KUKA KRL program: EPS_2_25694_WD05A_A_20260120031658.src

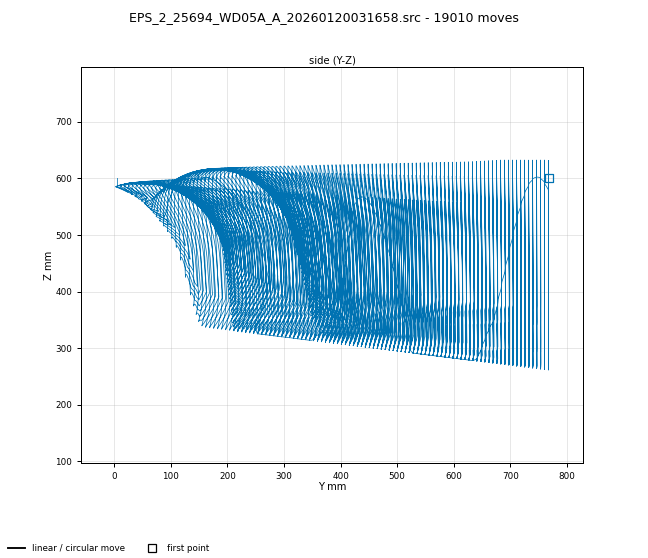
[picture p0: tool path of EPS_2_25694_WD05A_A_20260120031658.src, 19010 of 19012 moves have a stored position in this frame; points joined in program order, loops and branches not executed]
&ACCESS RVP
&REL 4
&COMMENT QRS 19112012
&PARAM EDITMASK = *
DEF PART()
EXT BAS (BAS_COMMAND :IN,REAL :IN )
INT I
BAS (#INITMOV,0 )

;KUKA QRS Post kuka4.cps  Date:22-06-2017 !

File_ID=3000

QRS_PRE_INIT()

;Init var - Until changes are made in qrs_pre_init
Outlet_Square_prg=0
Inlet_1_Square_prg=0
Inlet_2_Square_prg=0
Inlet_3_Square_prg=0
Inlet_4_Square_prg=0
Inlet_5_Square_prg=0

Outlet_1={X 0.000, Y 683.250, Z 507.000, B 0.000, E1 0.000 }
Inlet_1={X 0.000, Y 685.380, Z 477.000, B 0.000, E1 102.000 }
Inlet_2={X 0.000, Y 688.950, Z 427.000, B 0.000, E1 192.000 }
Outlet_1_type=251
Inlet_1_type=251
Inlet_2_type=251
;QRS#1=Sidecore dimensions
;QRS#2=250-10" PVC SDR 35
;QRS#3=250-10" PVC SDR 35
;QRS#4=250-10" PVC SDR 35
;QRS#5=
;QRS#6=
;QRS#7=
;QRS#8=
;QRS#9=14M PSX
;QRS#10=14M PSX
;QRS#11=14M PSX
;QRS#12=
;QRS#13=
;QRS#14=
;QRS#15=
;QRS#16=1524x152x991 3,25'
;QRS#17=EPS Height
;QRS#18=632,5
;QRS#19=*
;QRS#20= UPDATED VERSION 22-06-2017
;QRS#21=*
Outlet_Square=0100
Inlet_1_Square=0100
Inlet_2_Square=0100
Inlet_3_Square=0
Inlet_4_Square=0
Inlet_5_Square=0
Mill_Square=1
Outlet_Square_Prg=205
Inlet_1_Square_prg=205
Inlet_2_Square_prg=205

QRS_INIT()

$ADVANCE=5

; T1
PTP {E1 174.372,E2 174.372}
PTP {X 0,Y 767.508,A -85,B 0,C 180,E1 174.372,E2 174.372,E3 0,E4 0,E5 0,E6 0}
QRS_SPEED_INIT()
LIN {X 0,Y 767.508,Z 600,A -85,B 0,C 180,E1 174.372,E2 174.372,E3 0,E4 0,E5 0,E6 0} C_VEL
LIN {X 0,Y 767.508,Z 587.394,A -85,B 0,C 180,E1 174.372,E2 174.372} C_VEL
LIN {X 0,Y 767.508,Z 578.978,A -85,B 0,C 180,E1 174.372,E2 174.372} C_VEL
LIN {X 0,Y 767.496,Z 577.286,A -85,B 0,C 180,E1 174.143,E2 174.143} C_VEL
LIN {X 0,Y 767.495,Z 584.736,A -85,B 0,C 180,E1 173.186,E2 173.186} C_VEL
LIN {X 0,Y 767.498,Z 591.178,A -85,B 0,C 180,E1 172.132,E2 172.132} C_VEL
LIN {X 0,Y 767.492,Z 596.003,A -85,B 0,C 180,E1 171.075,E2 171.075} C_VEL
LIN {X 0,Y 767.497,Z 599.35,A -85,B 0,C 180,E1 170.014,E2 170.014} C_VEL
LIN {X 0,Y 767.492,Z 601.3,A -85,B 0,C 180,E1 168.951,E2 168.951} C_VEL
LIN {X 0,Y 767.498,Z 601.872,A -85,B 0,C 180,E1 167.883,E2 167.883} C_VEL
LIN {X 0,Y 767.495,Z 601.085,A -85,B 0,C 180,E1 166.811,E2 166.811} C_VEL
LIN {X 0,Y 767.497,Z 598.914,A -85,B 0,C 180,E1 165.735,E2 165.735} C_VEL
LIN {X 0,Y 767.496,Z 595.272,A -85,B 0,C 180,E1 164.653,E2 164.653} C_VEL
LIN {X 0,Y 767.496,Z 590.038,A -85,B 0,C 180,E1 163.566,E2 163.566} C_VEL
LIN {X 0,Y 767.497,Z 584.889,A -85,B 0,C 180,E1 162.746,E2 162.746} C_VEL
LIN {X 0,Y 767.497,Z 577.442,A -85,B 0,C 180,E1 161.786,E2 161.786} C_VEL
LIN {X 0,Y 767.497,Z 569.535,A -85,B 0,C 180,E1 160.958,E2 160.958} C_VEL
LIN {X 0,Y 767.498,Z 560.365,A -85,B 0,C 180,E1 160.16,E2 160.16} C_VEL
LIN {X 0,Y 767.498,Z 550.234,A -85,B 0,C 180,E1 159.429,E2 159.429} C_VEL
LIN {X 0,Y 767.498,Z 538.398,A -85,B 0,C 180,E1 158.729,E2 158.729} C_VEL
LIN {X 0,Y 767.475,Z 526.685,A -85,B 0,C 180,E1 158.163,E2 158.163} C_VEL
LIN {X 0,Y 767.49,Z 514.099,A -85,B 0,C 180,E1 157.673,E2 157.673} C_VEL
LIN {X 0,Y 767.495,Z 500.169,A -85,B 0,C 180,E1 157.255,E2 157.255} C_VEL
LIN {X 0,Y 767.49,Z 487.078,A -85,B 0,C 180,E1 156.967,E2 156.967} C_VEL
LIN {X 0,Y 767.49,Z 473.61,A -85,B 0,C 180,E1 156.769,E2 156.769} C_VEL
LIN {X 0,Y 767.47,Z 340.133,A -85,B 0,C 180,E1 155.5,E2 155.5} C_VEL
LIN {X 0,Y 767.459,Z 318.185,A -85,B 0,C 180,E1 153.141,E2 153.141} C_VEL
LIN {X 0,Y 767.478,Z 297.746,A -85,B 0,C 180,E1 150.923,E2 150.923} C_VEL
LIN {X 0,Y 767.488,Z 274.468,A -85,B 0,C 180,E1 148.366,E2 148.366} C_VEL
LIN {X 0,Y 767.445,Z 261.318,A -85,B 0,C 180,E1 146.893,E2 146.893} C_VEL
LIN {X 0,Y 767.439,Z 261.317,A -85,B 0,C 180,E1 144.9,E2 144.9} C_VEL
LIN {X 0,Y 767.432,Z 261.318,A -85,B 0,C 180,E1 142.959,E2 142.959} C_VEL
LIN {X 0,Y 767.427,Z 261.318,A -85,B 0,C 180,E1 140.879,E2 140.879} C_VEL
LIN {X 0,Y 767.421,Z 261.319,A -85,B 0,C 180,E1 138.916,E2 138.916} C_VEL
LIN {X 0,Y 767.423,Z 261.32,A -85,B 0,C 180,E1 136.8,E2 136.8} C_VEL
LIN {X 0,Y 767.441,Z 261.321,A -85,B 0,C 180,E1 134.61,E2 134.61} C_VEL
LIN {X 0,Y 767.488,Z 261.324,A -85,B 0,C 180,E1 132.333,E2 132.333} C_VEL
LIN {X 0,Y 767.43,Z 261.325,A -85,B 0,C 180,E1 129.943,E2 129.943} C_VEL
LIN {X 0,Y 767.411,Z 261.322,A -85,B 0,C 180,E1 127.701,E2 127.701} C_VEL
LIN {X 0,Y 767.415,Z 261.321,A -85,B 0,C 180,E1 125.676,E2 125.676} C_VEL
LIN {X 0,Y 767.426,Z 261.319,A -85,B 0,C 180,E1 123.833,E2 123.833} C_VEL
LIN {X 0,Y 767.433,Z 261.317,A -85,B 0,C 180,E1 121.916,E2 121.916} C_VEL
LIN {X 0,Y 767.433,Z 261.317,A -85,B 0,C 180,E1 119.879,E2 119.879} C_VEL
LIN {X 0,Y 767.438,Z 261.318,A -85,B 0,C 180,E1 117.709,E2 117.709} C_VEL
LIN {X 0,Y 767.47,Z 261.322,A -85,B 0,C 180,E1 115.373,E2 115.373} C_VEL
LIN {X 0,Y 767.49,Z 261.31,A -85,B 0,C 180,E1 112.814,E2 112.814} C_VEL
LIN {X 0,Y 767.465,Z 261.31,A -85,B 0,C 180,E1 110.294,E2 110.294} C_VEL
LIN {X 0,Y 767.463,Z 261.314,A -85,B 0,C 180,E1 108.079,E2 108.079} C_VEL
LIN {X 0,Y 767.477,Z 261.32,A -85,B 0,C 180,E1 105.891,E2 105.891} C_VEL
LIN {X 0,Y 767.491,Z 261.326,A -85,B 0,C 180,E1 103.728,E2 103.728} C_VEL
LIN {X 0,Y 767.477,Z 261.319,A -85,B 0,C 180,E1 101.584,E2 101.584} C_VEL
LIN {X 0,Y 767.466,Z 261.315,A -85,B 0,C 180,E1 99.457,E2 99.457} C_VEL
LIN {X 0,Y 767.463,Z 261.311,A -85,B 0,C 180,E1 97.342,E2 97.342} C_VEL
LIN {X 0,Y 767.466,Z 261.309,A -85,B 0,C 180,E1 95.238,E2 95.238} C_VEL
LIN {X 0,Y 767.488,Z 261.451,A -85,B 0,C 180,E1 94.68,E2 94.68} C_VEL
LIN {X 0,Y 767.448,Z 277.919,A -85,B 0,C 180,E1 92.355,E2 92.355} C_VEL
LIN {X 0,Y 767.478,Z 291.914,A -85,B 0,C 180,E1 90.393,E2 90.393} C_VEL
LIN {X 0,Y 767.487,Z 427.006,A -85,B 0,C 180,E1 89.103,E2 89.103} C_VEL
LIN {X 0,Y 767.496,Z 441.53,A -85,B 0,C 180,E1 88.857,E2 88.857} C_VEL
LIN {X 0,Y 767.491,Z 454.808,A -85,B 0,C 180,E1 88.53,E2 88.53} C_VEL
LIN {X 0,Y 767.491,Z 467.782,A -85,B 0,C 180,E1 88.105,E2 88.105} C_VEL
LIN {X 0,Y 767.489,Z 480.34,A -85,B 0,C 180,E1 87.582,E2 87.582} C_VEL
LIN {X 0,Y 767.499,Z 492.93,A -85,B 0,C 180,E1 86.928,E2 86.928} C_VEL
LIN {X 0,Y 767.497,Z 504.226,A -85,B 0,C 180,E1 86.208,E2 86.208} C_VEL
LIN {X 0,Y 767.496,Z 514.374,A -85,B 0,C 180,E1 85.421,E2 85.421} C_VEL
LIN {X 0,Y 767.498,Z 522.781,A -85,B 0,C 180,E1 84.634,E2 84.634} C_VEL
LIN {X 0,Y 767.497,Z 530.839,A -85,B 0,C 180,E1 83.714,E2 83.714} C_VEL
LIN {X 0,Y 767.498,Z 536.529,A -85,B 0,C 180,E1 82.924,E2 82.924} C_VEL
LIN {X 0,Y 767.499,Z 541.169,A -85,B 0,C 180,E1 82.133,E2 82.133} C_VEL
LIN {X 0,Y 767.498,Z 545.995,A -85,B 0,C 180,E1 81.076,E2 81.076} C_VEL
LIN {X 0,Y 767.493,Z 549.347,A -85,B 0,C 180,E1 80.016,E2 80.016} C_VEL
LIN {X 0,Y 767.491,Z 551.299,A -85,B 0,C 180,E1 78.952,E2 78.952} C_VEL
LIN {X 0,Y 767.497,Z 551.873,A -85,B 0,C 180,E1 77.885,E2 77.885} C_VEL
LIN {X 0,Y 767.495,Z 551.087,A -85,B 0,C 180,E1 76.813,E2 76.813} C_VEL
LIN {X 0,Y 767.49,Z 548.919,A -85,B 0,C 180,E1 75.736,E2 75.736} C_VEL
LIN {X 0,Y 767.492,Z 545.279,A -85,B 0,C 180,E1 74.654,E2 74.654} C_VEL
LIN {X 0,Y 767.496,Z 540.047,A -85,B 0,C 180,E1 73.567,E2 73.567} C_VEL
LIN {X 0,Y 767.498,Z 534.9,A -85,B 0,C 180,E1 72.748,E2 72.748} C_VEL
LIN {X 0,Y 767.497,Z 527.445,A -85,B 0,C 180,E1 71.786,E2 71.786} C_VEL
LIN {X 0,Y 767.496,Z 519.552,A -85,B 0,C 180,E1 70.959,E2 70.959} C_VEL
LIN {X 0,Y 767.498,Z 510.369,A -85,B 0,C 180,E1 70.16,E2 70.16} C_VEL
LIN {X 0,Y 767.498,Z 500.261,A -85,B 0,C 180,E1 69.431,E2 69.431} C_VEL
LIN {X 0,Y 767.498,Z 488.432,A -85,B 0,C 180,E1 68.731,E2 68.731} C_VEL
LIN {X 0,Y 767.482,Z 476.709,A -85,B 0,C 180,E1 68.164,E2 68.164} C_VEL
LIN {X 0,Y 767.474,Z 464.146,A -85,B 0,C 180,E1 67.675,E2 67.675} C_VEL
LIN {X 0,Y 767.496,Z 450.193,A -85,B 0,C 180,E1 67.255,E2 67.255} C_VEL
LIN {X 0,Y 767.466,Z 437.138,A -85,B 0,C 180,E1 66.968,E2 66.968} C_VEL
LIN {X 0,Y 767.451,Z 423.723,A -85,B 0,C 180,E1 66.77,E2 66.77} C_VEL
LIN {X 0,Y 767.496,Z 291.939,A -85,B 0,C 180,E1 65.521,E2 65.521} C_VEL
LIN {X 0,Y 767.491,Z 273.937,A -85,B 0,C 180,E1 62.997,E2 62.997} C_VEL
LIN {X 0,Y 767.45,Z 261.318,A -85,B 0,C 180,E1 61.185,E2 61.185} C_VEL
LIN {X 0,Y 767.434,Z 261.318,A -85,B 0,C 180,E1 59.087,E2 59.087} C_VEL
LIN {X 0,Y 767.412,Z 261.32,A -85,B 0,C 180,E1 56.797,E2 56.797} C_VEL
LIN {X 0,Y 767.416,Z 261.319,A -85,B 0,C 180,E1 54.901,E2 54.901} C_VEL
LIN {X 0,Y 767.417,Z 261.319,A -85,B 0,C 180,E1 52.96,E2 52.96} C_VEL
LIN {X 0,Y 767.413,Z 261.319,A -85,B 0,C 180,E1 50.88,E2 50.88} C_VEL
LIN {X 0,Y 767.414,Z 261.319,A -85,B 0,C 180,E1 48.918,E2 48.918} C_VEL
LIN {X 0,Y 767.411,Z 261.32,A -85,B 0,C 180,E1 46.902,E2 46.902} C_VEL
LIN {X 0,Y 767.44,Z 261.317,A -85,B 0,C 180,E1 45.352,E2 45.352} C_VEL
LIN {X 0,Y 767.424,Z 261.318,A -85,B 0,C 180,E1 43.2,E2 43.2} C_VEL
LIN {X 0,Y 767.417,Z 261.319,A -85,B 0,C 180,E1 41.084,E2 41.084} C_VEL
LIN {X 0,Y 767.416,Z 261.319,A -85,B 0,C 180,E1 39.034,E2 39.034} C_VEL
LIN {X 0,Y 767.416,Z 261.319,A -85,B 0,C 180,E1 37.042,E2 37.042} C_VEL
LIN {X 0,Y 767.426,Z 261.321,A -85,B 0,C 180,E1 34.774,E2 34.774} C_VEL
LIN {X 0,Y 767.448,Z 261.323,A -85,B 0,C 180,E1 32.581,E2 32.581} C_VEL
LIN {X 0,Y 767.48,Z 261.313,A -85,B 0,C 180,E1 29.89,E2 29.89} C_VEL
LIN {X 0,Y 767.446,Z 261.316,A -85,B 0,C 180,E1 27.714,E2 27.714} C_VEL
LIN {X 0,Y 767.422,Z 261.317,A -85,B 0,C 180,E1 25.37,E2 25.37} C_VEL
LIN {X 0,Y 767.439,Z 261.315,A -85,B 0,C 180,E1 23.678,E2 23.678} C_VEL
LIN {X 0,Y 767.471,Z 261.313,A -85,B 0,C 180,E1 21.974,E2 21.974} C_VEL
LIN {X 0,Y 767.44,Z 261.315,A -85,B 0,C 180,E1 19.737,E2 19.737} C_VEL
LIN {X 0,Y 767.423,Z 261.317,A -85,B 0,C 180,E1 17.53,E2 17.53} C_VEL
LIN {X 0,Y 767.449,Z 261.314,A -85,B 0,C 180,E1 15.891,E2 15.891} C_VEL
LIN {X 0,Y 767.429,Z 261.316,A -85,B 0,C 180,E1 13.728,E2 13.728} C_VEL
LIN {X 0,Y 767.47,Z 261.312,A -85,B 0,C 180,E1 12.117,E2 12.117} C_VEL
LIN {X 0,Y 767.449,Z 261.313,A -85,B 0,C 180,E1 9.986,E2 9.986} C_VEL
LIN {X 0,Y 767.435,Z 261.315,A -85,B 0,C 180,E1 7.869,E2 7.869} C_VEL
LIN {X 0,Y 767.425,Z 261.317,A -85,B 0,C 180,E1 5.762,E2 5.762} C_VEL
LIN {X 0,Y 767.463,Z 261.312,A -85,B 0,C 180,E1 4.187,E2 4.187} C_VEL
LIN {X 0,Y 767.447,Z 261.313,A -85,B 0,C 180,E1 2.092,E2 2.092} C_VEL
LIN {X 0,Y 767.438,Z 261.314,A -85,B 0,C 180,E1 0,E2 0} C_VEL
LIN {X 0,Y 767.431,Z 261.315,A -85,B 0,C 180,E1 -2.092,E2 -2.092} C_VEL
LIN {X 0,Y 767.428,Z 261.317,A -85,B 0,C 180,E1 -4.187,E2 -4.187} C_VEL
LIN {X 0,Y 767.43,Z 261.318,A -85,B 0,C 180,E1 -6.288,E2 -6.288} C_VEL
LIN {X 0,Y 767.436,Z 261.319,A -85,B 0,C 180,E1 -8.397,E2 -8.397} C_VEL
LIN {X 0,Y 767.448,Z 261.321,A -85,B 0,C 180,E1 -10.518,E2 -10.518} C_VEL
LIN {X 0,Y 767.495,Z 261.312,A -85,B 0,C 180,E1 -13.189,E2 -13.189} C_VEL
LIN {X 0,Y 767.483,Z 261.309,A -85,B 0,C 180,E1 -15.347,E2 -15.347} C_VEL
LIN {X 0,Y 767.455,Z 261.311,A -85,B 0,C 180,E1 -17.529,E2 -17.529} C_VEL
LIN {X 0,Y 767.432,Z 261.316,A -85,B 0,C 180,E1 -19.939,E2 -19.939} C_VEL
LIN {X 0,Y 767.433,Z 261.317,A -85,B 0,C 180,E1 -21.976,E2 -21.976} C_VEL
LIN {X 0,Y 767.447,Z 261.321,A -85,B 0,C 180,E1 -24.25,E2 -24.25} C_VEL
LIN {X 0,Y 767.484,Z 261.328,A -85,B 0,C 180,E1 -26.574,E2 -26.574} C_VEL
LIN {X 0,Y 767.496,Z 261.31,A -85,B 0,C 180,E1 -28.927,E2 -28.927} C_VEL
LIN {X 0,Y 767.453,Z 261.311,A -85,B 0,C 180,E1 -31.348,E2 -31.348} C_VEL
LIN {X 0,Y 767.464,Z 261.309,A -85,B 0,C 180,E1 -33.203,E2 -33.203} C_VEL
LIN {X 0,Y 767.472,Z 261.309,A -85,B 0,C 180,E1 -35.098,E2 -35.098} C_VEL
LIN {X 0,Y 767.441,Z 261.313,A -85,B 0,C 180,E1 -37.438,E2 -37.438} C_VEL
LIN {X 0,Y 767.437,Z 261.318,A -85,B 0,C 180,E1 -39.709,E2 -39.709} C_VEL
LIN {X 0,Y 767.442,Z 261.319,A -85,B 0,C 180,E1 -41.78,E2 -41.78} C_VEL
LIN {X 0,Y 767.454,Z 261.322,A -85,B 0,C 180,E1 -43.919,E2 -43.919} C_VEL
LIN {X 0,Y 767.482,Z 261.326,A -85,B 0,C 180,E1 -46.137,E2 -46.137} C_VEL
LIN {X 0,Y 767.468,Z 261.308,A -85,B 0,C 180,E1 -48.922,E2 -48.922} C_VEL
LIN {X 0,Y 767.459,Z 261.309,A -85,B 0,C 180,E1 -50.971,E2 -50.971} C_VEL
LIN {X 0,Y 767.457,Z 261.31,A -85,B 0,C 180,E1 -52.962,E2 -52.962} C_VEL
LIN {X 0,Y 767.44,Z 261.314,A -85,B 0,C 180,E1 -55.228,E2 -55.228} C_VEL
LIN {X 0,Y 767.445,Z 261.317,A -85,B 0,C 180,E1 -57.421,E2 -57.421} C_VEL
LIN {X 0,Y 767.481,Z 261.326,A -85,B 0,C 180,E1 -59.872,E2 -59.872} C_VEL
LIN {X 0,Y 767.487,Z 261.312,A -85,B 0,C 180,E1 -62.285,E2 -62.285} C_VEL
LIN {X 0,Y 767.472,Z 261.307,A -85,B 0,C 180,E1 -64.627,E2 -64.627} C_VEL
LIN {X 0,Y 767.448,Z 261.312,A -85,B 0,C 180,E1 -66.894,E2 -66.894} C_VEL
LIN {X 0,Y 767.444,Z 261.474,A -85,B 0,C 180,E1 -67.176,E2 -67.176} C_VEL
LIN {X 0,Y 767.477,Z 284.386,A -85,B 0,C 180,E1 -69.43,E2 -69.43} C_VEL
LIN {X 0,Y 767.461,Z 308.744,A -85,B 0,C 180,E1 -71.791,E2 -71.791} C_VEL
LIN {X 0,Y 767.489,Z 335.826,A -85,B 0,C 180,E1 -74.383,E2 -74.383} C_VEL
LIN {X 0,Y 767.49,Z 364.366,A -85,B 0,C 180,E1 -77.081,E2 -77.081} C_VEL
LIN {X 0,Y 767.489,Z 369.344,A -85,B 0,C 180,E1 -77.549,E2 -77.549} C_VEL
LIN {X 0,Y 767.475,Z 506.982,A -85,B 0,C 180,E1 -78.852,E2 -78.852} C_VEL
LIN {X 0,Y 767.49,Z 520.974,A -85,B 0,C 180,E1 -79.085,E2 -79.085} C_VEL
LIN {X 0,Y 767.479,Z 534.589,A -85,B 0,C 180,E1 -79.418,E2 -79.418} C_VEL
LIN {X 0,Y 767.474,Z 546.922,A -85,B 0,C 180,E1 -79.816,E2 -79.816} C_VEL
LIN {X 0,Y 767.483,Z 559.858,A -85,B 0,C 180,E1 -80.35,E2 -80.35} C_VEL
LIN {X 0,Y 767.499,Z 571.476,A -85,B 0,C 180,E1 -80.944,E2 -80.944} C_VEL
LIN {X 0,Y 767.496,Z 582.151,A -85,B 0,C 180,E1 -81.605,E2 -81.605} C_VEL
LIN {X 0,Y 767.498,Z 592.712,A -85,B 0,C 180,E1 -82.397,E2 -82.397} C_VEL
LIN {X 0,Y 767.497,Z 601.428,A -85,B 0,C 180,E1 -83.188,E2 -83.188} C_VEL
LIN {X 0,Y 767.496,Z 608.249,A -85,B 0,C 180,E1 -83.926,E2 -83.926} C_VEL
LIN {X 0,Y 767.497,Z 614.711,A -85,B 0,C 180,E1 -84.765,E2 -84.765} C_VEL
LIN {X 0,Y 767.494,Z 621.131,A -85,B 0,C 180,E1 -85.814,E2 -85.814} C_VEL
LIN {X 0,Y 767.496,Z 625.929,A -85,B 0,C 180,E1 -86.862,E2 -86.862} C_VEL
LIN {X 0,Y 767.496,Z 629.265,A -85,B 0,C 180,E1 -87.909,E2 -87.909} C_VEL
LIN {X 0,Y 767.497,Z 631.231,A -85,B 0,C 180,E1 -88.955,E2 -88.955} C_VEL
LIN {X 0,Y 767.494,Z 631.889,A -85,B 0,C 180,E1 -90.001,E2 -90.001} C_VEL
LIN {X 0,Y 767.497,Z 631.228,A -85,B 0,C 180,E1 -91.047,E2 -91.047} C_VEL
LIN {X 0,Y 767.496,Z 629.258,A -85,B 0,C 180,E1 -92.093,E2 -92.093} C_VEL
LIN {X 0,Y 767.496,Z 625.919,A -85,B 0,C 180,E1 -93.14,E2 -93.14} C_VEL
LIN {X 0,Y 767.494,Z 621.118,A -85,B 0,C 180,E1 -94.188,E2 -94.188} C_VEL
LIN {X 0,Y 767.497,Z 614.693,A -85,B 0,C 180,E1 -95.237,E2 -95.237} C_VEL
LIN {X 0,Y 767.496,Z 608.238,A -85,B 0,C 180,E1 -96.075,E2 -96.075} C_VEL
LIN {X 0,Y 767.498,Z 600.054,A -85,B 0,C 180,E1 -96.947,E2 -96.947} C_VEL
LIN {X 0,Y 767.497,Z 591.068,A -85,B 0,C 180,E1 -97.737,E2 -97.737} C_VEL
LIN {X 0,Y 767.498,Z 580.173,A -85,B 0,C 180,E1 -98.53,E2 -98.53} C_VEL
LIN {X 0,Y 767.498,Z 569.055,A -85,B 0,C 180,E1 -99.191,E2 -99.191} C_VEL
LIN {X 0,Y 767.494,Z 556.885,A -85,B 0,C 180,E1 -99.783,E2 -99.783} C_VEL
LIN {X 0,Y 767.472,Z 544.967,A -85,B 0,C 180,E1 -100.253,E2 -100.253} C_VEL
LIN {X 0,Y 767.484,Z 532.071,A -85,B 0,C 180,E1 -100.651,E2 -100.651} C_VEL
LIN {X 0,Y 767.487,Z 519.13,A -85,B 0,C 180,E1 -100.951,E2 -100.951} C_VEL
LIN {X 0,Y 767.474,Z 505.285,A -85,B 0,C 180,E1 -101.167,E2 -101.167} C_VEL
LIN {X 0,Y 767.488,Z 369.199,A -85,B 0,C 180,E1 -102.465,E2 -102.465} C_VEL
LIN {X 0,Y 767.498,Z 342.937,A -85,B 0,C 180,E1 -104.942,E2 -104.942} C_VEL
LIN {X 0,Y 767.479,Z 315.807,A -85,B 0,C 180,E1 -107.529,E2 -107.529} C_VEL
LIN {X 0,Y 767.465,Z 289.028,A -85,B 0,C 180,E1 -110.117,E2 -110.117} C_VEL
LIN {X 0,Y 767.459,Z 264.333,A -85,B 0,C 180,E1 -112.541,E2 -112.541} C_VEL
LIN {X 0,Y 767.444,Z 261.317,A -85,B 0,C 180,E1 -112.844,E2 -112.844} C_VEL
LIN {X 0,Y 767.44,Z 261.316,A -85,B 0,C 180,E1 -114.826,E2 -114.826} C_VEL
LIN {X 0,Y 767.442,Z 261.319,A -85,B 0,C 180,E1 -116.567,E2 -116.567} C_VEL
LIN {X 0,Y 767.45,Z 261.321,A -85,B 0,C 180,E1 -118.334,E2 -118.334} C_VEL
LIN {X 0,Y 767.461,Z 261.323,A -85,B 0,C 180,E1 -120.132,E2 -120.132} C_VEL
LIN {X 0,Y 767.471,Z 261.324,A -85,B 0,C 180,E1 -121.962,E2 -121.962} C_VEL
LIN {X 0,Y 767.47,Z 261.325,A -85,B 0,C 180,E1 -123.847,E2 -123.847} C_VEL
LIN {X 0,Y 767.478,Z 261.325,A -85,B 0,C 180,E1 -125.74,E2 -125.74} C_VEL
LIN {X 0,Y 767.469,Z 261.325,A -85,B 0,C 180,E1 -127.698,E2 -127.698} C_VEL
LIN {X 0,Y 767.422,Z 261.324,A -85,B 0,C 180,E1 -129.942,E2 -129.942} C_VEL
LIN {X 0,Y 767.427,Z 261.325,A -85,B 0,C 180,E1 -131.782,E2 -131.782} C_VEL
LIN {X 0,Y 767.405,Z 261.325,A -85,B 0,C 180,E1 -133.923,E2 -133.923} C_VEL
LIN {X 0,Y 767.401,Z 261.323,A -85,B 0,C 180,E1 -136.077,E2 -136.077} C_VEL
LIN {X 0,Y 767.406,Z 261.323,A -85,B 0,C 180,E1 -138.218,E2 -138.218} C_VEL
LIN {X 0,Y 767.411,Z 261.321,A -85,B 0,C 180,E1 -140.059,E2 -140.059} C_VEL
LIN {X 0,Y 767.426,Z 261.319,A -85,B 0,C 180,E1 -141.716,E2 -141.716} C_VEL
LIN {X 0,Y 767.434,Z 261.317,A -85,B 0,C 180,E1 -143.611,E2 -143.611} C_VEL
LIN {X 0,Y 767.44,Z 261.315,A -85,B 0,C 180,E1 -145.537,E2 -145.537} C_VEL
LIN {X 0,Y 767.449,Z 261.314,A -85,B 0,C 180,E1 -147.419,E2 -147.419} C_VEL
LIN {X 0,Y 767.465,Z 261.311,A -85,B 0,C 180,E1 -149.263,E2 -149.263} C_VEL
LIN {X 0,Y 767.472,Z 261.309,A -85,B 0,C 180,E1 -151.183,E2 -151.183} C_VEL
LIN {X 0,Y 767.45,Z 261.312,A -85,B 0,C 180,E1 -153.437,E2 -153.437} C_VEL
LIN {X 0,Y 767.451,Z 261.318,A -85,B 0,C 180,E1 -155.751,E2 -155.751} C_VEL
LIN {X 0,Y 767.483,Z 261.323,A -85,B 0,C 180,E1 -158.026,E2 -158.026} C_VEL
LIN {X 0,Y 767.487,Z 261.319,A -85,B 0,C 180,E1 -160.264,E2 -160.264} C_VEL
LIN {X 0,Y 767.48,Z 261.311,A -85,B 0,C 180,E1 -162.472,E2 -162.472} C_VEL
LIN {X 0,Y 767.491,Z 261.304,A -85,B 0,C 180,E1 -164.653,E2 -164.653} C_VEL
LIN {X 0,Y 767.489,Z 261.303,A -85,B 0,C 180,E1 -166.811,E2 -166.811} C_VEL
LIN {X 0,Y 767.481,Z 261.322,A -85,B 0,C 180,E1 -169.483,E2 -169.483} C_VEL
LIN {X 0,Y 767.478,Z 261.447,A -85,B 0,C 180,E1 -171.008,E2 -171.008} C_VEL
LIN {X 0,Y 767.457,Z 283.481,A -85,B 0,C 180,E1 -173.449,E2 -173.449} C_VEL
LIN {X 0,Y 767.459,Z 303.894,A -85,B 0,C 180,E1 -175.682,E2 -175.682} C_VEL
LIN {X 0,Y 767.479,Z 326.891,A -85,B 0,C 180,E1 -178.169,E2 -178.169} C_VEL
LIN {X 0,Y 767.492,Z 340.14,A -85,B 0,C 180,E1 -179.591,E2 -179.591} C_VEL
LIN {X 0,Y 767.473,Z 477.124,A -85,B 0,C 180,E1 -180.899,E2 -180.899} C_VEL
LIN {X 0,Y 767.479,Z 491.605,A -85,B 0,C 180,E1 -181.144,E2 -181.144} C_VEL
LIN {X 0,Y 767.493,Z 504.85,A -85,B 0,C 180,E1 -181.471,E2 -181.471} C_VEL
LIN {X 0,Y 767.473,Z 517.827,A -85,B 0,C 180,E1 -181.896,E2 -181.896} C_VEL
LIN {X 0,Y 767.487,Z 530.368,A -85,B 0,C 180,E1 -182.419,E2 -182.419} C_VEL
LIN {X 0,Y 767.499,Z 542.953,A -85,B 0,C 180,E1 -183.073,E2 -183.073} C_VEL
LIN {X 0,Y 767.497,Z 554.246,A -85,B 0,C 180,E1 -183.794,E2 -183.794} C_VEL
LIN {X 0,Y 767.496,Z 564.389,A -85,B 0,C 180,E1 -184.58,E2 -184.58} C_VEL
LIN {X 0,Y 767.498,Z 572.794,A -85,B 0,C 180,E1 -185.368,E2 -185.368} C_VEL
LIN {X 0,Y 767.496,Z 577.286,A -85,B 0,C 180,E1 -185.857,E2 -185.857} C_VEL
LIN {X 0,Y 766.835,Z 580.572,A -85,B 0,C 180,E1 -186.229,E2 -186.229} C_VEL
LIN {X 0,Y 763.971,Z 585.532,A -85,B 0,C 180,E1 -186.84,E2 -186.84} C_VEL
LIN {X 0,Y 761.109,Z 589.729,A -85,B 0,C 180,E1 -187.476,E2 -187.476} C_VEL
LIN {X 0,Y 760.438,Z 591.975,A -85,B 0,C 180,E1 -187.881,E2 -187.881} C_VEL
LIN {X 0,Y 760.444,Z 595.945,A -85,B 0,C 180,E1 -188.742,E2 -188.742} C_VEL
LIN {X 0,Y 760.422,Z 599.305,A -85,B 0,C 180,E1 -189.731,E2 -189.731} C_VEL
LIN {X 0,Y 760.417,Z 601.287,A -85,B 0,C 180,E1 -190.616,E2 -190.616} C_VEL
LIN {X 0,Y 760.446,Z 602.402,A -85,B 0,C 180,E1 -191.691,E2 -191.691} C_VEL
LIN {X 0,Y 760.439,Z 602.159,A -85,B 0,C 180,E1 -192.772,E2 -192.772} C_VEL
LIN {X 0,Y 760.42,Z 600.537,A -85,B 0,C 180,E1 -193.857,E2 -193.857} C_VEL
LIN {X 0,Y 760.447,Z 597.472,A -85,B 0,C 180,E1 -194.946,E2 -194.946} C_VEL
LIN {X 0,Y 760.431,Z 592.858,A -85,B 0,C 180,E1 -196.042,E2 -196.042} C_VEL
LIN {X 0,Y 760.448,Z 588.36,A -85,B 0,C 180,E1 -196.844,E2 -196.844} C_VEL
LIN {X 0,Y 760.456,Z 581.463,A -85,B 0,C 180,E1 -197.834,E2 -197.834} C_VEL
LIN {X 0,Y 760.447,Z 572.963,A -85,B 0,C 180,E1 -198.807,E2 -198.807} C_VEL
LIN {X 0,Y 760.456,Z 563.937,A -85,B 0,C 180,E1 -199.645,E2 -199.645} C_VEL
LIN {X 0,Y 760.486,Z 554.782,A -85,B 0,C 180,E1 -200.356,E2 -200.356} C_VEL
LIN {X 0,Y 760.473,Z 544.026,A -85,B 0,C 180,E1 -201.052,E2 -201.052} C_VEL
LIN {X 0,Y 760.488,Z 532.055,A -85,B 0,C 180,E1 -201.689,E2 -201.689} C_VEL
LIN {X 0,Y 760.5,Z 518.772,A -85,B 0,C 180,E1 -202.258,E2 -202.258} C_VEL
LIN {X 0,Y 760.523,Z 506.057,A -85,B 0,C 180,E1 -202.685,E2 -202.685} C_VEL
LIN {X 0,Y 760.539,Z 491.807,A -85,B 0,C 180,E1 -203.045,E2 -203.045} C_VEL
LIN {X 0,Y 760.549,Z 477.909,A -85,B 0,C 180,E1 -203.284,E2 -203.284} C_VEL
LIN {X 0,Y 760.452,Z 340.316,A -85,B 0,C 180,E1 -204.614,E2 -204.614} C_VEL
LIN {X 0,Y 760.453,Z 318.478,A -85,B 0,C 180,E1 -206.977,E2 -206.977} C_VEL
LIN {X 0,Y 760.497,Z 299.436,A -85,B 0,C 180,E1 -209.058,E2 -209.058} C_VEL
LIN {X 0,Y 760.532,Z 277.263,A -85,B 0,C 180,E1 -211.511,E2 -211.511} C_VEL
LIN {X 0,Y 760.433,Z 262.316,A -85,B 0,C 180,E1 -213.203,E2 -213.203} C_VEL
LIN {X 0,Y 760.421,Z 262.315,A -85,B 0,C 180,E1 -215.472,E2 -215.472} C_VEL
LIN {X 0,Y 760.447,Z 262.313,A -85,B 0,C 180,E1 -217.613,E2 -217.613} C_VEL
LIN {X 0,Y 760.454,Z 262.323,A -85,B 0,C 180,E1 -220.148,E2 -220.148} C_VEL
LIN {X 0,Y 760.417,Z 262.318,A -85,B 0,C 180,E1 -222.531,E2 -222.531} C_VEL
LIN {X 0,Y 760.393,Z 262.321,A -85,B 0,C 180,E1 -224.434,E2 -224.434} C_VEL
LIN {X 0,Y 760.393,Z 262.318,A -85,B 0,C 180,E1 -226.695,E2 -226.695} C_VEL
LIN {X 0,Y 760.397,Z 262.318,A -85,B 0,C 180,E1 -228.452,E2 -228.452} C_VEL
LIN {X 0,Y 760.369,Z 262.321,A -85,B 0,C 180,E1 -230.696,E2 -230.696} C_VEL
LIN {X 0,Y 760.375,Z 262.32,A -85,B 0,C 180,E1 -232.555,E2 -232.555} C_VEL
LIN {X 0,Y 760.387,Z 262.319,A -85,B 0,C 180,E1 -234.525,E2 -234.525} C_VEL
LIN {X 0,Y 760.442,Z 262.318,A -85,B 0,C 180,E1 -236.951,E2 -236.951} C_VEL
LIN {X 0,Y 760.433,Z 262.317,A -85,B 0,C 180,E1 -239.561,E2 -239.561} C_VEL
LIN {X 0,Y 760.426,Z 262.314,A -85,B 0,C 180,E1 -241.98,E2 -241.98} C_VEL
LIN {X 0,Y 760.445,Z 262.312,A -85,B 0,C 180,E1 -243.759,E2 -243.759} C_VEL
LIN {X 0,Y 760.418,Z 262.316,A -85,B 0,C 180,E1 -246.089,E2 -246.089} C_VEL
LIN {X 0,Y 760.451,Z 262.32,A -85,B 0,C 180,E1 -248.482,E2 -248.482} C_VEL
LIN {X 0,Y 760.454,Z 262.321,A -85,B 0,C 180,E1 -250.634,E2 -250.634} C_VEL
LIN {X 0,Y 760.463,Z 262.314,A -85,B 0,C 180,E1 -252.857,E2 -252.857} C_VEL
LIN {X 0,Y 760.488,Z 262.306,A -85,B 0,C 180,E1 -255.262,E2 -255.262} C_VEL
LIN {X 0,Y 760.471,Z 262.313,A -85,B 0,C 180,E1 -257.768,E2 -257.768} C_VEL
LIN {X 0,Y 760.457,Z 262.318,A -85,B 0,C 180,E1 -260.251,E2 -260.251} C_VEL
LIN {X 0,Y 760.433,Z 262.314,A -85,B 0,C 180,E1 -262.59,E2 -262.59} C_VEL
LIN {X 0,Y 760.442,Z 262.312,A -85,B 0,C 180,E1 -264.714,E2 -264.714} C_VEL
LIN {X 0,Y 760.483,Z 262.368,A -85,B 0,C 180,E1 -265.277,E2 -265.277} C_VEL
LIN {X 0,Y 760.434,Z 280.746,A -85,B 0,C 180,E1 -267.887,E2 -267.887} C_VEL
LIN {X 0,Y 760.455,Z 292.23,A -85,B 0,C 180,E1 -269.504,E2 -269.504} C_VEL
LIN {X 0,Y 760.533,Z 428.035,A -85,B 0,C 180,E1 -270.807,E2 -270.807} C_VEL
LIN {X 0,Y 760.546,Z 442.227,A -85,B 0,C 180,E1 -271.054,E2 -271.054} C_VEL
LIN {X 0,Y 760.505,Z 456.48,A -85,B 0,C 180,E1 -271.417,E2 -271.417} C_VEL
LIN {X 0,Y 760.501,Z 469.136,A -85,B 0,C 180,E1 -271.846,E2 -271.846} C_VEL
LIN {X 0,Y 760.491,Z 481.494,A -85,B 0,C 180,E1 -272.374,E2 -272.374} C_VEL
LIN {X 0,Y 760.474,Z 493.961,A -85,B 0,C 180,E1 -273.035,E2 -273.035} C_VEL
LIN {X 0,Y 760.461,Z 504.215,A -85,B 0,C 180,E1 -273.695,E2 -273.695} C_VEL
LIN {X 0,Y 760.478,Z 514.465,A -85,B 0,C 180,E1 -274.489,E2 -274.489} C_VEL
LIN {X 0,Y 760.445,Z 522.969,A -85,B 0,C 180,E1 -275.284,E2 -275.284} C_VEL
LIN {X 0,Y 760.452,Z 531.026,A -85,B 0,C 180,E1 -276.199,E2 -276.199} C_VEL
LIN {X 0,Y 760.443,Z 537.724,A -85,B 0,C 180,E1 -277.142,E2 -277.142} C_VEL
LIN {X 0,Y 760.445,Z 543.596,A -85,B 0,C 180,E1 -278.207,E2 -278.207} C_VEL
LIN {X 0,Y 760.448,Z 547.001,A -85,B 0,C 180,E1 -279.007,E2 -279.007} C_VEL
LIN {X 0,Y 760.421,Z 550.213,A -85,B 0,C 180,E1 -280.078,E2 -280.078} C_VEL
LIN {X 0,Y 760.432,Z 552.012,A -85,B 0,C 180,E1 -281.152,E2 -281.152} C_VEL
LIN {X 0,Y 760.43,Z 552.452,A -85,B 0,C 180,E1 -282.23,E2 -282.23} C_VEL
LIN {X 0,Y 760.43,Z 551.525,A -85,B 0,C 180,E1 -283.312,E2 -283.312} C_VEL
LIN {X 0,Y 760.419,Z 549.195,A -85,B 0,C 180,E1 -284.399,E2 -284.399} C_VEL
LIN {X 0,Y 760.449,Z 545.375,A -85,B 0,C 180,E1 -285.491,E2 -285.491} C_VEL
LIN {X 0,Y 760.441,Z 541.411,A -85,B 0,C 180,E1 -286.314,E2 -286.314} C_VEL
LIN {X 0,Y 760.431,Z 536.46,A -85,B 0,C 180,E1 -287.141,E2 -287.141} C_VEL
LIN {X 0,Y 760.446,Z 529.22,A -85,B 0,C 180,E1 -288.11,E2 -288.11} C_VEL
LIN {X 0,Y 760.464,Z 521.562,A -85,B 0,C 180,E1 -288.944,E2 -288.944} C_VEL
LIN {X 0,Y 760.452,Z 512.245,A -85,B 0,C 180,E1 -289.784,E2 -289.784} C_VEL
LIN {X 0,Y 760.47,Z 501.87,A -85,B 0,C 180,E1 -290.556,E2 -290.556} C_VEL
LIN {X 0,Y 760.481,Z 490.379,A -85,B 0,C 180,E1 -291.262,E2 -291.262} C_VEL
LIN {X 0,Y 760.476,Z 477.5,A -85,B 0,C 180,E1 -291.901,E2 -291.901} C_VEL
LIN {X 0,Y 760.484,Z 464.93,A -85,B 0,C 180,E1 -292.399,E2 -292.399} C_VEL
LIN {X 0,Y 760.534,Z 451.893,A -85,B 0,C 180,E1 -292.803,E2 -292.803} C_VEL
LIN {X 0,Y 760.497,Z 438.047,A -85,B 0,C 180,E1 -293.12,E2 -293.12} C_VEL
LIN {X 0,Y 760.499,Z 424.267,A -85,B 0,C 180,E1 -293.329,E2 -293.329} C_VEL
LIN {X 0,Y 760.481,Z 292.176,A -85,B 0,C 180,E1 -294.593,E2 -294.593} C_VEL
LIN {X 0,Y 760.476,Z 274.24,A -85,B 0,C 180,E1 -297.123,E2 -297.123} C_VEL
LIN {X 0,Y 760.426,Z 262.317,A -85,B 0,C 180,E1 -298.831,E2 -298.831} C_VEL
LIN {X 0,Y 760.402,Z 262.317,A -85,B 0,C 180,E1 -301.055,E2 -301.055} C_VEL
LIN {X 0,Y 760.409,Z 262.316,A -85,B 0,C 180,E1 -303.045,E2 -303.045} C_VEL
LIN {X 0,Y 760.4,Z 262.317,A -85,B 0,C 180,E1 -304.933,E2 -304.933} C_VEL
LIN {X 0,Y 760.422,Z 262.316,A -85,B 0,C 180,E1 -306.777,E2 -306.777} C_VEL
LIN {X 0,Y 760.423,Z 262.315,A -85,B 0,C 180,E1 -308.78,E2 -308.78} C_VEL
LIN {X 0,Y 760.412,Z 262.315,A -85,B 0,C 180,E1 -310.946,E2 -310.946} C_VEL
LIN {X 0,Y 760.398,Z 262.317,A -85,B 0,C 180,E1 -312.97,E2 -312.97} C_VEL
LIN {X 0,Y 760.401,Z 262.316,A -85,B 0,C 180,E1 -315.174,E2 -315.174} C_VEL
LIN {X 0,Y 760.416,Z 262.318,A -85,B 0,C 180,E1 -317.466,E2 -317.466} C_VEL
LIN {X 0,Y 760.453,Z 262.322,A -85,B 0,C 180,E1 -319.86,E2 -319.86} C_VEL
LIN {X 0,Y 760.408,Z 262.316,A -85,B 0,C 180,E1 -322.558,E2 -322.558} C_VEL
LIN {X 0,Y 760.409,Z 262.316,A -85,B 0,C 180,E1 -324.527,E2 -324.527} C_VEL
LIN {X 0,Y 760.438,Z 262.313,A -85,B 0,C 180,E1 -326.45,E2 -326.45} C_VEL
LIN {X 0,Y 760.443,Z 262.313,A -85,B 0,C 180,E1 -328.33,E2 -328.33} C_VEL
LIN {X 0,Y 760.401,Z 262.316,A -85,B 0,C 180,E1 -330.777,E2 -330.777} C_VEL
LIN {X 0,Y 760.416,Z 262.314,A -85,B 0,C 180,E1 -332.576,E2 -332.576} C_VEL
LIN {X 0,Y 760.398,Z 262.317,A -85,B 0,C 180,E1 -334.515,E2 -334.515} C_VEL
LIN {X 0,Y 760.433,Z 262.315,A -85,B 0,C 180,E1 -336.091,E2 -336.091} C_VEL
LIN {X 0,Y 760.401,Z 262.316,A -85,B 0,C 180,E1 -338.485,E2 -338.485} C_VEL
LIN {X 0,Y 760.405,Z 262.316,A -85,B 0,C 180,E1 -340.633,E2 -340.633} C_VEL
LIN {X 0,Y 760.416,Z 262.315,A -85,B 0,C 180,E1 -342.304,E2 -342.304} C_VEL
LIN {X 0,Y 760.412,Z 262.315,A -85,B 0,C 180,E1 -344.506,E2 -344.506} C_VEL
LIN {X 0,Y 760.395,Z 262.318,A -85,B 0,C 180,E1 -346.686,E2 -346.686} C_VEL
LIN {X 0,Y 760.4,Z 262.316,A -85,B 0,C 180,E1 -348.308,E2 -348.308} C_VEL
LIN {X 0,Y 760.413,Z 262.315,A -85,B 0,C 180,E1 -350.456,E2 -350.456} C_VEL
LIN {X 0,Y 760.398,Z 262.318,A -85,B 0,C 180,E1 -352.59,E2 -352.59} C_VEL
LIN {X 0,Y 760.413,Z 262.318,A -85,B 0,C 180,E1 -354.715,E2 -354.715} C_VEL
LIN {X 0,Y 760.473,Z 262.316,A -85,B 0,C 180,E1 -357.36,E2 -357.36} C_VEL
LIN {X 0,Y 760.435,Z 262.312,A -85,B 0,C 180,E1 -360,E2 -360} C_VEL
LIN {X 0,Y 760.419,Z 262.314,A -85,B 0,C 180,E1 -362.112,E2 -362.112} C_VEL
LIN {X 0,Y 760.406,Z 262.316,A -85,B 0,C 180,E1 -364.226,E2 -364.226} C_VEL
LIN {X 0,Y 760.436,Z 262.312,A -85,B 0,C 180,E1 -365.869,E2 -365.869} C_VEL
LIN {X 0,Y 760.406,Z 262.315,A -85,B 0,C 180,E1 -367.942,E2 -367.942} C_VEL
LIN {X 0,Y 760.401,Z 262.316,A -85,B 0,C 180,E1 -370.08,E2 -370.08} C_VEL
LIN {X 0,Y 760.429,Z 262.314,A -85,B 0,C 180,E1 -372.231,E2 -372.231} C_VEL
LIN {X 0,Y 760.469,Z 262.319,A -85,B 0,C 180,E1 -374.741,E2 -374.741} C_VEL
LIN {X 0,Y 760.454,Z 262.315,A -85,B 0,C 180,E1 -377.142,E2 -377.142} C_VEL
LIN {X 0,Y 760.442,Z 262.313,A -85,B 0,C 180,E1 -379.366,E2 -379.366} C_VEL
LIN {X 0,Y 760.413,Z 262.315,A -85,B 0,C 180,E1 -381.62,E2 -381.62} C_VEL
LIN {X 0,Y 760.447,Z 262.312,A -85,B 0,C 180,E1 -383.333,E2 -383.333} C_VEL
LIN {X 0,Y 760.434,Z 262.312,A -85,B 0,C 180,E1 -385.653,E2 -385.653} C_VEL
LIN {X 0,Y 760.436,Z 262.315,A -85,B 0,C 180,E1 -388.019,E2 -388.019} C_VEL
LIN {X 0,Y 760.434,Z 262.324,A -85,B 0,C 180,E1 -390.438,E2 -390.438} C_VEL
LIN {X 0,Y 760.456,Z 262.311,A -85,B 0,C 180,E1 -393.055,E2 -393.055} C_VEL
LIN {X 0,Y 760.412,Z 262.314,A -85,B 0,C 180,E1 -395.473,E2 -395.473} C_VEL
LIN {X 0,Y 760.425,Z 262.314,A -85,B 0,C 180,E1 -397.615,E2 -397.615} C_VEL
LIN {X 0,Y 760.434,Z 262.312,A -85,B 0,C 180,E1 -399.462,E2 -399.462} C_VEL
LIN {X 0,Y 760.412,Z 262.318,A -85,B 0,C 180,E1 -401.747,E2 -401.747} C_VEL
LIN {X 0,Y 760.425,Z 262.323,A -85,B 0,C 180,E1 -404.074,E2 -404.074} C_VEL
LIN {X 0,Y 760.463,Z 262.312,A -85,B 0,C 180,E1 -406.69,E2 -406.69} C_VEL
LIN {X 0,Y 760.419,Z 262.314,A -85,B 0,C 180,E1 -409.159,E2 -409.159} C_VEL
LIN {X 0,Y 760.438,Z 262.312,A -85,B 0,C 180,E1 -411.221,E2 -411.221} C_VEL
LIN {X 0,Y 760.424,Z 262.314,A -85,B 0,C 180,E1 -413.262,E2 -413.262} C_VEL
LIN {X 0,Y 760.438,Z 262.321,A -85,B 0,C 180,E1 -415.817,E2 -415.817} C_VEL
LIN {X 0,Y 760.467,Z 262.313,A -85,B 0,C 180,E1 -418.333,E2 -418.333} C_VEL
LIN {X 0,Y 760.434,Z 262.312,A -85,B 0,C 180,E1 -420.78,E2 -420.78} C_VEL
LIN {X 0,Y 760.453,Z 262.311,A -85,B 0,C 180,E1 -422.58,E2 -422.58} C_VEL
LIN {X 0,Y 760.42,Z 262.314,A -85,B 0,C 180,E1 -424.932,E2 -424.932} C_VEL
LIN {X 0,Y 760.449,Z 262.488,A -85,B 0,C 180,E1 -427.055,E2 -427.055} C_VEL
LIN {X 0,Y 760.586,Z 277.458,A -85,B 0,C 180,E1 -428.551,E2 -428.551} C_VEL
LIN {X 0,Y 760.528,Z 301.551,A -85,B 0,C 180,E1 -430.918,E2 -430.918} C_VEL
LIN {X 0,Y 760.526,Z 326.171,A -85,B 0,C 180,E1 -433.304,E2 -433.304} C_VEL
LIN {X 0,Y 760.493,Z 351.616,A -85,B 0,C 180,E1 -435.738,E2 -435.738} C_VEL
LIN {X 0,Y 760.487,Z 369.528,A -85,B 0,C 180,E1 -437.435,E2 -437.435} C_VEL
LIN {X 0,Y 760.512,Z 507.129,A -85,B 0,C 180,E1 -438.749,E2 -438.749} C_VEL
LIN {X 0,Y 760.519,Z 521.1,A -85,B 0,C 180,E1 -438.984,E2 -438.984} C_VEL
LIN {X 0,Y 760.502,Z 534.725,A -85,B 0,C 180,E1 -439.32,E2 -439.32} C_VEL
LIN {X 0,Y 760.478,Z 547.078,A -85,B 0,C 180,E1 -439.722,E2 -439.722} C_VEL
LIN {X 0,Y 760.496,Z 559.507,A -85,B 0,C 180,E1 -440.235,E2 -440.235} C_VEL
LIN {X 0,Y 760.495,Z 571.71,A -85,B 0,C 180,E1 -440.86,E2 -440.86} C_VEL
LIN {X 0,Y 760.462,Z 582.428,A -85,B 0,C 180,E1 -441.527,E2 -441.527} C_VEL
LIN {X 0,Y 760.453,Z 593.041,A -85,B 0,C 180,E1 -442.326,E2 -442.326} C_VEL
LIN {X 0,Y 760.465,Z 601.808,A -85,B 0,C 180,E1 -443.124,E2 -443.124} C_VEL
LIN {X 0,Y 760.444,Z 609.326,A -85,B 0,C 180,E1 -443.947,E2 -443.947} C_VEL
LIN {X 0,Y 760.435,Z 615.182,A -85,B 0,C 180,E1 -444.716,E2 -444.716} C_VEL
LIN {X 0,Y 760.435,Z 621.651,A -85,B 0,C 180,E1 -445.775,E2 -445.775} C_VEL
LIN {X 0,Y 760.425,Z 626.489,A -85,B 0,C 180,E1 -446.833,E2 -446.833} C_VEL
LIN {X 0,Y 760.424,Z 629.854,A -85,B 0,C 180,E1 -447.89,E2 -447.89} C_VEL
LIN {X 0,Y 760.451,Z 631.837,A -85,B 0,C 180,E1 -448.946,E2 -448.946} C_VEL
LIN {X 0,Y 760.438,Z 632.5,A -85,B 0,C 180,E1 -450.001,E2 -450.001} C_VEL
LIN {X 0,Y 760.451,Z 631.833,A -85,B 0,C 180,E1 -451.057,E2 -451.057} C_VEL
LIN {X 0,Y 760.424,Z 629.846,A -85,B 0,C 180,E1 -452.113,E2 -452.113} C_VEL
LIN {X 0,Y 760.425,Z 626.479,A -85,B 0,C 180,E1 -453.169,E2 -453.169} C_VEL
LIN {X 0,Y 760.435,Z 621.637,A -85,B 0,C 180,E1 -454.227,E2 -454.227} C_VEL
LIN {X 0,Y 760.436,Z 615.164,A -85,B 0,C 180,E1 -455.286,E2 -455.286} C_VEL
LIN {X 0,Y 760.454,Z 608.076,A -85,B 0,C 180,E1 -456.201,E2 -456.201} C_VEL
LIN {X 0,Y 760.448,Z 600.427,A -85,B 0,C 180,E1 -457.011,E2 -457.011} C_VEL
LIN {X 0,Y 760.474,Z 591.389,A -85,B 0,C 180,E1 -457.809,E2 -457.809} C_VEL
LIN {X 0,Y 760.471,Z 580.441,A -85,B 0,C 180,E1 -458.609,E2 -458.609} C_VEL
LIN {X 0,Y 760.491,Z 569.279,A -85,B 0,C 180,E1 -459.277,E2 -459.277} C_VEL
LIN {X 0,Y 760.5,Z 557.748,A -85,B 0,C 180,E1 -459.845,E2 -459.845} C_VEL
LIN {X 0,Y 760.484,Z 545.122,A -85,B 0,C 180,E1 -460.348,E2 -460.348} C_VEL
LIN {X 0,Y 760.531,Z 532.21,A -85,B 0,C 180,E1 -460.75,E2 -460.75} C_VEL
LIN {X 0,Y 760.531,Z 518.355,A -85,B 0,C 180,E1 -461.069,E2 -461.069} C_VEL
LIN {X 0,Y 760.512,Z 503.948,A -85,B 0,C 180,E1 -461.288,E2 -461.288} C_VEL
LIN {X 0,Y 760.514,Z 369.826,A -85,B 0,C 180,E1 -462.562,E2 -462.562} C_VEL
LIN {X 0,Y 760.491,Z 367.322,A -85,B 0,C 180,E1 -462.772,E2 -462.772} C_VEL
LIN {X 0,Y 760.505,Z 340.145,A -85,B 0,C 180,E1 -465.356,E2 -465.356} C_VEL
LIN {X 0,Y 760.552,Z 314.397,A -85,B 0,C 180,E1 -467.833,E2 -467.833} C_VEL
LIN {X 0,Y 760.544,Z 288.57,A -85,B 0,C 180,E1 -470.354,E2 -470.354} C_VEL
LIN {X 0,Y 760.573,Z 265.763,A -85,B 0,C 180,E1 -472.613,E2 -472.613} C_VEL
LIN {X 0,Y 760.426,Z 262.316,A -85,B 0,C 180,E1 -472.967,E2 -472.967} C_VEL
LIN {X 0,Y 760.415,Z 262.315,A -85,B 0,C 180,E1 -475.071,E2 -475.071} C_VEL
LIN {X 0,Y 760.455,Z 262.313,A -85,B 0,C 180,E1 -477.423,E2 -477.423} C_VEL
LIN {X 0,Y 760.454,Z 262.32,A -85,B 0,C 180,E1 -480.023,E2 -480.023} C_VEL
LIN {X 0,Y 760.411,Z 262.318,A -85,B 0,C 180,E1 -482.295,E2 -482.295} C_VEL
LIN {X 0,Y 760.421,Z 262.318,A -85,B 0,C 180,E1 -484.187,E2 -484.187} C_VEL
LIN {X 0,Y 760.417,Z 262.318,A -85,B 0,C 180,E1 -486.124,E2 -486.124} C_VEL
LIN {X 0,Y 760.409,Z 262.318,A -85,B 0,C 180,E1 -488.11,E2 -488.11} C_VEL
LIN {X 0,Y 760.391,Z 262.319,A -85,B 0,C 180,E1 -490.153,E2 -490.153} C_VEL
LIN {X 0,Y 760.369,Z 262.321,A -85,B 0,C 180,E1 -492.259,E2 -492.259} C_VEL
LIN {X 0,Y 760.372,Z 262.321,A -85,B 0,C 180,E1 -494.067,E2 -494.067} C_VEL
LIN {X 0,Y 760.396,Z 262.318,A -85,B 0,C 180,E1 -496.301,E2 -496.301} C_VEL
LIN {X 0,Y 760.41,Z 262.318,A -85,B 0,C 180,E1 -498.454,E2 -498.454} C_VEL
LIN {X 0,Y 760.443,Z 262.319,A -85,B 0,C 180,E1 -500.69,E2 -500.69} C_VEL
LIN {X 0,Y 760.443,Z 262.316,A -85,B 0,C 180,E1 -503.261,E2 -503.261} C_VEL
LIN {X 0,Y 760.421,Z 262.314,A -85,B 0,C 180,E1 -505.814,E2 -505.814} C_VEL
LIN {X 0,Y 760.409,Z 262.317,A -85,B 0,C 180,E1 -507.936,E2 -507.936} C_VEL
LIN {X 0,Y 760.424,Z 262.317,A -85,B 0,C 180,E1 -509.982,E2 -509.982} C_VEL
LIN {X 0,Y 760.447,Z 262.318,A -85,B 0,C 180,E1 -512.161,E2 -512.161} C_VEL
LIN {X 0,Y 760.473,Z 262.316,A -85,B 0,C 180,E1 -514.509,E2 -514.509} C_VEL
LIN {X 0,Y 760.439,Z 262.312,A -85,B 0,C 180,E1 -517.24,E2 -517.24} C_VEL
LIN {X 0,Y 760.448,Z 262.313,A -85,B 0,C 180,E1 -519.512,E2 -519.512} C_VEL
LIN {X 0,Y 760.457,Z 262.318,A -85,B 0,C 180,E1 -521.75,E2 -521.75} C_VEL
LIN {X 0,Y 760.445,Z 262.323,A -85,B 0,C 180,E1 -523.959,E2 -523.959} C_VEL
LIN {X 0,Y 760.445,Z 262.317,A -85,B 0,C 180,E1 -526.144,E2 -526.144} C_VEL
LIN {X 0,Y 760.444,Z 262.314,A -85,B 0,C 180,E1 -528.308,E2 -528.308} C_VEL
LIN {X 0,Y 760.476,Z 262.31,A -85,B 0,C 180,E1 -530.891,E2 -530.891} C_VEL
LIN {X 0,Y 760.525,Z 280.96,A -85,B 0,C 180,E1 -532.991,E2 -532.991} C_VEL
LIN {X 0,Y 760.497,Z 302.583,A -85,B 0,C 180,E1 -535.377,E2 -535.377} C_VEL
LIN {X 0,Y 760.47,Z 325.62,A -85,B 0,C 180,E1 -537.889,E2 -537.889} C_VEL
LIN {X 0,Y 760.478,Z 340.452,A -85,B 0,C 180,E1 -539.489,E2 -539.489} C_VEL
LIN {X 0,Y 760.528,Z 476.936,A -85,B 0,C 180,E1 -540.792,E2 -540.792} C_VEL
LIN {X 0,Y 760.531,Z 491.549,A -85,B 0,C 180,E1 -541.039,E2 -541.039} C_VEL
LIN {X 0,Y 760.508,Z 505.42,A -85,B 0,C 180,E1 -541.385,E2 -541.385} C_VEL
LIN {X 0,Y 760.486,Z 519.17,A -85,B 0,C 180,E1 -541.847,E2 -541.847} C_VEL
LIN {X 0,Y 760.489,Z 531.518,A -85,B 0,C 180,E1 -542.375,E2 -542.375} C_VEL
LIN {X 0,Y 760.474,Z 543.989,A -85,B 0,C 180,E1 -543.036,E2 -543.036} C_VEL
LIN {X 0,Y 760.462,Z 554.241,A -85,B 0,C 180,E1 -543.697,E2 -543.697} C_VEL
LIN {X 0,Y 760.479,Z 564.486,A -85,B 0,C 180,E1 -544.49,E2 -544.49} C_VEL
LIN {X 0,Y 760.446,Z 572.984,A -85,B 0,C 180,E1 -545.285,E2 -545.285} C_VEL
LIN {X 0,Y 760.454,Z 581.037,A -85,B 0,C 180,E1 -546.2,E2 -546.2} C_VEL
LIN {X 0,Y 760.445,Z 587.734,A -85,B 0,C 180,E1 -547.143,E2 -547.143} C_VEL
LIN {X 0,Y 760.438,Z 591.975,A -85,B 0,C 180,E1 -547.881,E2 -547.881} C_VEL
LIN {X 0,Y 759.764,Z 594.062,A -85,B 0,C 180,E1 -548.294,E2 -548.294} C_VEL
LIN {X 0,Y 756.879,Z 596.94,A -85,B 0,C 180,E1 -548.978,E2 -548.978} C_VEL
LIN {X 0,Y 754.447,Z 598.829,A -85,B 0,C 180,E1 -549.536,E2 -549.536} C_VEL
LIN {X 0,Y 753.404,Z 600.001,A -85,B 0,C 180,E1 -549.97,E2 -549.97} C_VEL
LIN {X 0,Y 753.32,Z 600.315,A -85,B 0,C 180,E1 -550.118,E2 -550.118} C_VEL
LIN {X 0,Y 753.331,Z 602.116,A -85,B 0,C 180,E1 -551.26,E2 -551.26} C_VEL
LIN {X 0,Y 753.337,Z 602.418,A -85,B 0,C 180,E1 -552.348,E2 -552.348} C_VEL
LIN {X 0,Y 753.329,Z 601.357,A -85,B 0,C 180,E1 -553.441,E2 -553.441} C_VEL
LIN {X 0,Y 753.337,Z 598.881,A -85,B 0,C 180,E1 -554.539,E2 -554.539} C_VEL
LIN {X 0,Y 753.361,Z 594.875,A -85,B 0,C 180,E1 -555.642,E2 -555.642} C_VEL
LIN {X 0,Y 753.359,Z 589.307,A -85,B 0,C 180,E1 -556.732,E2 -556.732} C_VEL
LIN {X 0,Y 753.358,Z 582.676,A -85,B 0,C 180,E1 -557.728,E2 -557.728} C_VEL
LIN {X 0,Y 753.393,Z 574.436,A -85,B 0,C 180,E1 -558.712,E2 -558.712} C_VEL
LIN {X 0,Y 753.387,Z 565.793,A -85,B 0,C 180,E1 -559.554,E2 -559.554} C_VEL
LIN {X 0,Y 753.436,Z 555.216,A -85,B 0,C 180,E1 -560.403,E2 -560.403} C_VEL
LIN {X 0,Y 753.447,Z 544.403,A -85,B 0,C 180,E1 -561.115,E2 -561.115} C_VEL
LIN {X 0,Y 753.484,Z 532.583,A -85,B 0,C 180,E1 -561.754,E2 -561.754} C_VEL
LIN {X 0,Y 753.483,Z 521.181,A -85,B 0,C 180,E1 -562.26,E2 -562.26} C_VEL
LIN {X 0,Y 753.524,Z 507.977,A -85,B 0,C 180,E1 -562.727,E2 -562.727} C_VEL
LIN {X 0,Y 753.564,Z 493.126,A -85,B 0,C 180,E1 -563.119,E2 -563.119} C_VEL
LIN {X 0,Y 753.579,Z 478.791,A -85,B 0,C 180,E1 -563.377,E2 -563.377} C_VEL
LIN {X 0,Y 753.6,Z 448.634,A -85,B 0,C 180,E1 -563.685,E2 -563.685} C_VEL
LIN {X 0,Y 753.478,Z 340.721,A -85,B 0,C 180,E1 -564.717,E2 -564.717} C_VEL
LIN {X 0,Y 753.424,Z 338.99,A -85,B 0,C 180,E1 -564.878,E2 -564.878} C_VEL
LIN {X 0,Y 753.457,Z 317.303,A -85,B 0,C 180,E1 -567.248,E2 -567.248} C_VEL
LIN {X 0,Y 753.514,Z 297.859,A -85,B 0,C 180,E1 -569.396,E2 -569.396} C_VEL
LIN {X 0,Y 753.617,Z 274.655,A -85,B 0,C 180,E1 -571.991,E2 -571.991} C_VEL
LIN {X 0,Y 753.4,Z 263.194,A -85,B 0,C 180,E1 -573.296,E2 -573.296} C_VEL
LIN {X 0,Y 753.404,Z 263.192,A -85,B 0,C 180,E1 -575.854,E2 -575.854} C_VEL
LIN {X 0,Y 753.416,Z 263.192,A -85,B 0,C 180,E1 -577.85,E2 -577.85} C_VEL
LIN {X 0,Y 753.383,Z 263.2,A -85,B 0,C 180,E1 -580.325,E2 -580.325} C_VEL
LIN {X 0,Y 753.383,Z 263.192,A -85,B 0,C 180,E1 -582.743,E2 -582.743} C_VEL
LIN {X 0,Y 753.336,Z 263.197,A -85,B 0,C 180,E1 -585.037,E2 -585.037} C_VEL
LIN {X 0,Y 753.384,Z 263.194,A -85,B 0,C 180,E1 -587.264,E2 -587.264} C_VEL
LIN {X 0,Y 753.364,Z 263.206,A -85,B 0,C 180,E1 -589.676,E2 -589.676} C_VEL
LIN {X 0,Y 753.372,Z 263.194,A -85,B 0,C 180,E1 -592.212,E2 -592.212} C_VEL
LIN {X 0,Y 753.363,Z 263.195,A -85,B 0,C 180,E1 -594.143,E2 -594.143} C_VEL
LIN {X 0,Y 753.371,Z 263.193,A -85,B 0,C 180,E1 -596.092,E2 -596.092} C_VEL
LIN {X 0,Y 753.386,Z 263.192,A -85,B 0,C 180,E1 -597.997,E2 -597.997} C_VEL
LIN {X 0,Y 753.387,Z 263.193,A -85,B 0,C 180,E1 -600.477,E2 -600.477} C_VEL
LIN {X 0,Y 753.441,Z 263.191,A -85,B 0,C 180,E1 -603.186,E2 -603.186} C_VEL
LIN {X 0,Y 753.39,Z 263.191,A -85,B 0,C 180,E1 -605.852,E2 -605.852} C_VEL
LIN {X 0,Y 753.393,Z 263.193,A -85,B 0,C 180,E1 -608.167,E2 -608.167} C_VEL
LIN {X 0,Y 753.402,Z 263.199,A -85,B 0,C 180,E1 -610.445,E2 -610.445} C_VEL
LIN {X 0,Y 753.422,Z 263.194,A -85,B 0,C 180,E1 -612.692,E2 -612.692} C_VEL
LIN {X 0,Y 753.437,Z 263.185,A -85,B 0,C 180,E1 -615.207,E2 -615.207} C_VEL
LIN {X 0,Y 753.417,Z 263.19,A -85,B 0,C 180,E1 -617.652,E2 -617.652} C_VEL
LIN {X 0,Y 753.414,Z 263.196,A -85,B 0,C 180,E1 -620.223,E2 -620.223} C_VEL
LIN {X 0,Y 753.408,Z 263.191,A -85,B 0,C 180,E1 -622.52,E2 -622.52} C_VEL
LIN {X 0,Y 753.394,Z 263.191,A -85,B 0,C 180,E1 -624.664,E2 -624.664} C_VEL
LIN {X 0,Y 753.46,Z 263.293,A -85,B 0,C 180,E1 -625.249,E2 -625.249} C_VEL
LIN {X 0,Y 753.399,Z 281.554,A -85,B 0,C 180,E1 -627.868,E2 -627.868} C_VEL
LIN {X 0,Y 753.412,Z 292.216,A -85,B 0,C 180,E1 -629.383,E2 -629.383} C_VEL
LIN {X 0,Y 753.661,Z 312.348,A -85,B 0,C 180,E1 -629.583,E2 -629.583} C_VEL
LIN {X 0,Y 753.568,Z 427.714,A -85,B 0,C 180,E1 -630.698,E2 -630.698} C_VEL
LIN {X 0,Y 753.589,Z 442.06,A -85,B 0,C 180,E1 -630.947,E2 -630.947} C_VEL
LIN {X 0,Y 753.513,Z 456.921,A -85,B 0,C 180,E1 -631.33,E2 -631.33} C_VEL
LIN {X 0,Y 753.506,Z 470.334,A -85,B 0,C 180,E1 -631.797,E2 -631.797} C_VEL
LIN {X 0,Y 753.489,Z 482.457,A -85,B 0,C 180,E1 -632.33,E2 -632.33} C_VEL
LIN {X 0,Y 753.456,Z 493.607,A -85,B 0,C 180,E1 -632.929,E2 -632.929} C_VEL
LIN {X 0,Y 753.407,Z 503.921,A -85,B 0,C 180,E1 -633.597,E2 -633.597} C_VEL
LIN {X 0,Y 753.414,Z 514.212,A -85,B 0,C 180,E1 -634.398,E2 -634.398} C_VEL
LIN {X 0,Y 753.388,Z 522.757,A -85,B 0,C 180,E1 -635.2,E2 -635.2} C_VEL
LIN {X 0,Y 753.373,Z 530.975,A -85,B 0,C 180,E1 -636.136,E2 -636.136} C_VEL
LIN {X 0,Y 753.358,Z 536.732,A -85,B 0,C 180,E1 -636.941,E2 -636.941} C_VEL
LIN {X 0,Y 753.342,Z 542.877,A -85,B 0,C 180,E1 -638.016,E2 -638.016} C_VEL
LIN {X 0,Y 753.351,Z 547.385,A -85,B 0,C 180,E1 -639.093,E2 -639.093} C_VEL
LIN {X 0,Y 753.317,Z 550.446,A -85,B 0,C 180,E1 -640.174,E2 -640.174} C_VEL
LIN {X 0,Y 753.33,Z 552.111,A -85,B 0,C 180,E1 -641.258,E2 -641.258} C_VEL
LIN {X 0,Y 753.335,Z 552.419,A -85,B 0,C 180,E1 -642.347,E2 -642.347} C_VEL
LIN {X 0,Y 753.334,Z 551.358,A -85,B 0,C 180,E1 -643.44,E2 -643.44} C_VEL
LIN {X 0,Y 753.334,Z 548.886,A -85,B 0,C 180,E1 -644.538,E2 -644.538} C_VEL
LIN {X 0,Y 753.364,Z 544.872,A -85,B 0,C 180,E1 -645.641,E2 -645.641} C_VEL
LIN {X 0,Y 753.357,Z 540.841,A -85,B 0,C 180,E1 -646.463,E2 -646.463} C_VEL
LIN {X 0,Y 753.369,Z 535.665,A -85,B 0,C 180,E1 -647.307,E2 -647.307} C_VEL
LIN {X 0,Y 753.365,Z 528.226,A -85,B 0,C 180,E1 -648.286,E2 -648.286} C_VEL
LIN {X 0,Y 753.375,Z 520.344,A -85,B 0,C 180,E1 -649.13,E2 -649.13} C_VEL
LIN {X 0,Y 753.401,Z 510.787,A -85,B 0,C 180,E1 -649.977,E2 -649.977} C_VEL
LIN {X 0,Y 753.431,Z 500.105,A -85,B 0,C 180,E1 -650.757,E2 -650.757} C_VEL
LIN {X 0,Y 753.477,Z 488.317,A -85,B 0,C 180,E1 -651.46,E2 -651.46} C_VEL
LIN {X 0,Y 753.466,Z 476.345,A -85,B 0,C 180,E1 -652.043,E2 -652.043} C_VEL
LIN {X 0,Y 753.491,Z 463.468,A -85,B 0,C 180,E1 -652.546,E2 -652.546} C_VEL
LIN {X 0,Y 753.535,Z 450.413,A -85,B 0,C 180,E1 -652.942,E2 -652.942} C_VEL
LIN {X 0,Y 753.546,Z 436.758,A -85,B 0,C 180,E1 -653.247,E2 -653.247} C_VEL
LIN {X 0,Y 753.527,Z 423.027,A -85,B 0,C 180,E1 -653.449,E2 -653.449} C_VEL
LIN {X 0,Y 753.618,Z 293.433,A -85,B 0,C 180,E1 -654.689,E2 -654.689} C_VEL
LIN {X 0,Y 753.426,Z 292.154,A -85,B 0,C 180,E1 -654.716,E2 -654.716} C_VEL
LIN {X 0,Y 753.426,Z 273.33,A -85,B 0,C 180,E1 -657.397,E2 -657.397} C_VEL
LIN {X 0,Y 753.387,Z 263.194,A -85,B 0,C 180,E1 -658.871,E2 -658.871} C_VEL
LIN {X 0,Y 753.36,Z 263.194,A -85,B 0,C 180,E1 -661.375,E2 -661.375} C_VEL
LIN {X 0,Y 753.373,Z 263.198,A -85,B 0,C 180,E1 -663.905,E2 -663.905} C_VEL
LIN {X 0,Y 753.377,Z 263.197,A -85,B 0,C 180,E1 -666.513,E2 -666.513} C_VEL
LIN {X 0,Y 753.391,Z 263.193,A -85,B 0,C 180,E1 -668.651,E2 -668.651} C_VEL
LIN {X 0,Y 753.381,Z 263.191,A -85,B 0,C 180,E1 -671.306,E2 -671.306} C_VEL
LIN {X 0,Y 753.371,Z 263.195,A -85,B 0,C 180,E1 -673.514,E2 -673.514} C_VEL
LIN {X 0,Y 753.378,Z 263.199,A -85,B 0,C 180,E1 -675.789,E2 -675.789} C_VEL
LIN {X 0,Y 753.39,Z 263.201,A -85,B 0,C 180,E1 -678.051,E2 -678.051} C_VEL
LIN {X 0,Y 753.393,Z 263.191,A -85,B 0,C 180,E1 -680.501,E2 -680.501} C_VEL
LIN {X 0,Y 753.376,Z 263.192,A -85,B 0,C 180,E1 -683.086,E2 -683.086} C_VEL
LIN {X 0,Y 753.368,Z 263.197,A -85,B 0,C 180,E1 -685.448,E2 -685.448} C_VEL
LIN {X 0,Y 753.417,Z 263.194,A -85,B 0,C 180,E1 -688,E2 -688} C_VEL
LIN {X 0,Y 753.387,Z 263.191,A -85,B 0,C 180,E1 -690.478,E2 -690.478} C_VEL
LIN {X 0,Y 753.358,Z 263.194,A -85,B 0,C 180,E1 -692.897,E2 -692.897} C_VEL
LIN {X 0,Y 753.389,Z 263.196,A -85,B 0,C 180,E1 -695.268,E2 -695.268} C_VEL
LIN {X 0,Y 753.405,Z 263.201,A -85,B 0,C 180,E1 -697.593,E2 -697.593} C_VEL
LIN {X 0,Y 753.417,Z 263.191,A -85,B 0,C 180,E1 -699.88,E2 -699.88} C_VEL
LIN {X 0,Y 753.38,Z 263.192,A -85,B 0,C 180,E1 -702.133,E2 -702.133} C_VEL
LIN {X 0,Y 753.388,Z 263.19,A -85,B 0,C 180,E1 -704.358,E2 -704.358} C_VEL
LIN {X 0,Y 753.35,Z 263.195,A -85,B 0,C 180,E1 -706.559,E2 -706.559} C_VEL
LIN {X 0,Y 753.383,Z 263.193,A -85,B 0,C 180,E1 -708.741,E2 -708.741} C_VEL
LIN {X 0,Y 753.395,Z 263.194,A -85,B 0,C 180,E1 -710.906,E2 -710.906} C_VEL
LIN {X 0,Y 753.405,Z 263.193,A -85,B 0,C 180,E1 -713.594,E2 -713.594} C_VEL
LIN {X 0,Y 753.418,Z 263.189,A -85,B 0,C 180,E1 -715.735,E2 -715.735} C_VEL
LIN {X 0,Y 753.399,Z 263.189,A -85,B 0,C 180,E1 -717.869,E2 -717.869} C_VEL
LIN {X 0,Y 753.39,Z 263.19,A -85,B 0,C 180,E1 -720,E2 -720} C_VEL
LIN {X 0,Y 753.383,Z 263.19,A -85,B 0,C 180,E1 -722.131,E2 -722.131} C_VEL
LIN {X 0,Y 753.387,Z 263.191,A -85,B 0,C 180,E1 -724.266,E2 -724.266} C_VEL
LIN {X 0,Y 753.383,Z 263.193,A -85,B 0,C 180,E1 -726.406,E2 -726.406} C_VEL
LIN {X 0,Y 753.371,Z 263.197,A -85,B 0,C 180,E1 -728.555,E2 -728.555} C_VEL
LIN {X 0,Y 753.417,Z 263.195,A -85,B 0,C 180,E1 -730.716,E2 -730.716} C_VEL
LIN {X 0,Y 753.404,Z 263.19,A -85,B 0,C 180,E1 -733.44,E2 -733.44} C_VEL
LIN {X 0,Y 753.403,Z 263.188,A -85,B 0,C 180,E1 -735.641,E2 -735.641} C_VEL
LIN {X 0,Y 753.371,Z 263.192,A -85,B 0,C 180,E1 -737.868,E2 -737.868} C_VEL
LIN {X 0,Y 753.398,Z 263.191,A -85,B 0,C 180,E1 -740.12,E2 -740.12} C_VEL
LIN {X 0,Y 753.394,Z 263.196,A -85,B 0,C 180,E1 -742.407,E2 -742.407} C_VEL
LIN {X 0,Y 753.405,Z 263.199,A -85,B 0,C 180,E1 -744.732,E2 -744.732} C_VEL
LIN {X 0,Y 753.415,Z 263.189,A -85,B 0,C 180,E1 -747.1,E2 -747.1} C_VEL
LIN {X 0,Y 753.385,Z 263.19,A -85,B 0,C 180,E1 -749.522,E2 -749.522} C_VEL
LIN {X 0,Y 753.388,Z 263.19,A -85,B 0,C 180,E1 -751.376,E2 -751.376} C_VEL
LIN {X 0,Y 753.401,Z 263.189,A -85,B 0,C 180,E1 -753.266,E2 -753.266} C_VEL
LIN {X 0,Y 753.393,Z 263.189,A -85,B 0,C 180,E1 -755.2,E2 -755.2} C_VEL
LIN {X 0,Y 753.396,Z 263.189,A -85,B 0,C 180,E1 -757.18,E2 -757.18} C_VEL
LIN {X 0,Y 753.388,Z 263.19,A -85,B 0,C 180,E1 -759.499,E2 -759.499} C_VEL
LIN {X 0,Y 753.382,Z 263.198,A -85,B 0,C 180,E1 -762.021,E2 -762.021} C_VEL
LIN {X 0,Y 753.389,Z 263.202,A -85,B 0,C 180,E1 -764.287,E2 -764.287} C_VEL
LIN {X 0,Y 753.414,Z 263.193,A -85,B 0,C 180,E1 -766.533,E2 -766.533} C_VEL
LIN {X 0,Y 753.409,Z 263.188,A -85,B 0,C 180,E1 -768.856,E2 -768.856} C_VEL
LIN {X 0,Y 753.388,Z 263.191,A -85,B 0,C 180,E1 -771.35,E2 -771.35} C_VEL
LIN {X 0,Y 753.374,Z 263.194,A -85,B 0,C 180,E1 -773.487,E2 -773.487} C_VEL
LIN {X 0,Y 753.409,Z 263.199,A -85,B 0,C 180,E1 -776.097,E2 -776.097} C_VEL
LIN {X 0,Y 753.393,Z 263.191,A -85,B 0,C 180,E1 -778.627,E2 -778.627} C_VEL
LIN {X 0,Y 753.399,Z 263.189,A -85,B 0,C 180,E1 -781.091,E2 -781.091} C_VEL
LIN {X 0,Y 753.382,Z 263.196,A -85,B 0,C 180,E1 -783.497,E2 -783.497} C_VEL
LIN {X 0,Y 753.415,Z 263.2,A -85,B 0,C 180,E1 -785.856,E2 -785.856} C_VEL
LIN {X 0,Y 753.435,Z 263.396,A -85,B 0,C 180,E1 -786.921,E2 -786.921} C_VEL
LIN {X 0,Y 753.717,Z 271.512,A -85,B 0,C 180,E1 -787.749,E2 -787.749} C_VEL
LIN {X 0,Y 753.65,Z 297.26,A -85,B 0,C 180,E1 -790.313,E2 -790.313} C_VEL
LIN {X 0,Y 753.544,Z 323.15,A -85,B 0,C 180,E1 -792.85,E2 -792.85} C_VEL
LIN {X 0,Y 753.513,Z 350.185,A -85,B 0,C 180,E1 -795.466,E2 -795.466} C_VEL
LIN {X 0,Y 753.474,Z 369.432,A -85,B 0,C 180,E1 -797.309,E2 -797.309} C_VEL
LIN {X 0,Y 753.654,Z 387.719,A -85,B 0,C 180,E1 -797.493,E2 -797.493} C_VEL
LIN {X 0,Y 753.554,Z 507.128,A -85,B 0,C 180,E1 -798.643,E2 -798.643} C_VEL
LIN {X 0,Y 753.558,Z 521.857,A -85,B 0,C 180,E1 -798.898,E2 -798.898} C_VEL
LIN {X 0,Y 753.533,Z 535.844,A -85,B 0,C 180,E1 -799.253,E2 -799.253} C_VEL
LIN {X 0,Y 753.476,Z 548.826,A -85,B 0,C 180,E1 -799.693,E2 -799.693} C_VEL
LIN {X 0,Y 753.466,Z 561.621,A -85,B 0,C 180,E1 -800.244,E2 -800.244} C_VEL
LIN {X 0,Y 753.449,Z 574.026,A -85,B 0,C 180,E1 -800.908,E2 -800.908} C_VEL
LIN {X 0,Y 753.412,Z 584.362,A -85,B 0,C 180,E1 -801.582,E2 -801.582} C_VEL
LIN {X 0,Y 753.401,Z 594.654,A -85,B 0,C 180,E1 -802.388,E2 -802.388} C_VEL
LIN {X 0,Y 753.389,Z 603.151,A -85,B 0,C 180,E1 -803.194,E2 -803.194} C_VEL
LIN {X 0,Y 753.385,Z 611.274,A -85,B 0,C 180,E1 -804.131,E2 -804.131} C_VEL
LIN {X 0,Y 753.376,Z 616.989,A -85,B 0,C 180,E1 -804.934,E2 -804.934} C_VEL
LIN {X 0,Y 753.339,Z 621.651,A -85,B 0,C 180,E1 -805.736,E2 -805.736} C_VEL
LIN {X 0,Y 753.354,Z 626.49,A -85,B 0,C 180,E1 -806.803,E2 -806.803} C_VEL
LIN {X 0,Y 753.324,Z 629.854,A -85,B 0,C 180,E1 -807.87,E2 -807.87} C_VEL
LIN {X 0,Y 753.351,Z 631.838,A -85,B 0,C 180,E1 -808.936,E2 -808.936} C_VEL
LIN {X 0,Y 753.339,Z 632.5,A -85,B 0,C 180,E1 -810.001,E2 -810.001} C_VEL
LIN {X 0,Y 753.351,Z 631.834,A -85,B 0,C 180,E1 -811.067,E2 -811.067} C_VEL
LIN {X 0,Y 753.324,Z 629.847,A -85,B 0,C 180,E1 -812.133,E2 -812.133} C_VEL
LIN {X 0,Y 753.354,Z 626.479,A -85,B 0,C 180,E1 -813.199,E2 -813.199} C_VEL
LIN {X 0,Y 753.339,Z 621.637,A -85,B 0,C 180,E1 -814.267,E2 -814.267} C_VEL
LIN {X 0,Y 753.358,Z 615.165,A -85,B 0,C 180,E1 -815.336,E2 -815.336} C_VEL
LIN {X 0,Y 753.371,Z 607.965,A -85,B 0,C 180,E1 -816.273,E2 -816.273} C_VEL
LIN {X 0,Y 753.394,Z 599.069,A -85,B 0,C 180,E1 -817.212,E2 -817.212} C_VEL
LIN {X 0,Y 753.412,Z 589.732,A -85,B 0,C 180,E1 -818.017,E2 -818.017} C_VEL
LIN {X 0,Y 753.435,Z 578.334,A -85,B 0,C 180,E1 -818.825,E2 -818.825} C_VEL
LIN {X 0,Y 753.476,Z 566.735,A -85,B 0,C 180,E1 -819.499,E2 -819.499} C_VEL
LIN {X 0,Y 753.501,Z 553.763,A -85,B 0,C 180,E1 -820.11,E2 -820.11} C_VEL
LIN {X 0,Y 753.51,Z 540.201,A -85,B 0,C 180,E1 -820.614,E2 -820.614} C_VEL
LIN {X 0,Y 753.579,Z 526.285,A -85,B 0,C 180,E1 -821.003,E2 -821.003} C_VEL
LIN {X 0,Y 753.579,Z 512.666,A -85,B 0,C 180,E1 -821.274,E2 -821.274} C_VEL
LIN {X 0,Y 753.573,Z 497.439,A -85,B 0,C 180,E1 -821.461,E2 -821.461} C_VEL
LIN {X 0,Y 753.512,Z 369.835,A -85,B 0,C 180,E1 -822.68,E2 -822.68} C_VEL
LIN {X 0,Y 753.477,Z 368.327,A -85,B 0,C 180,E1 -822.797,E2 -822.797} C_VEL
LIN {X 0,Y 753.512,Z 341.575,A -85,B 0,C 180,E1 -825.364,E2 -825.364} C_VEL
LIN {X 0,Y 753.583,Z 315.827,A -85,B 0,C 180,E1 -827.863,E2 -827.863} C_VEL
LIN {X 0,Y 753.646,Z 291.655,A -85,B 0,C 180,E1 -830.242,E2 -830.242} C_VEL
LIN {X 0,Y 753.711,Z 267.193,A -85,B 0,C 180,E1 -832.686,E2 -832.686} C_VEL
LIN {X 0,Y 753.407,Z 263.193,A -85,B 0,C 180,E1 -833.115,E2 -833.115} C_VEL
LIN {X 0,Y 753.437,Z 263.189,A -85,B 0,C 180,E1 -835.607,E2 -835.607} C_VEL
LIN {X 0,Y 753.392,Z 263.195,A -85,B 0,C 180,E1 -838.305,E2 -838.305} C_VEL
LIN {X 0,Y 753.387,Z 263.191,A -85,B 0,C 180,E1 -840.755,E2 -840.755} C_VEL
LIN {X 0,Y 753.41,Z 263.191,A -85,B 0,C 180,E1 -843.267,E2 -843.267} C_VEL
LIN {X 0,Y 753.38,Z 263.196,A -85,B 0,C 180,E1 -846.014,E2 -846.014} C_VEL
LIN {X 0,Y 753.408,Z 263.194,A -85,B 0,C 180,E1 -847.851,E2 -847.851} C_VEL
LIN {X 0,Y 753.337,Z 263.197,A -85,B 0,C 180,E1 -850.321,E2 -850.321} C_VEL
LIN {X 0,Y 753.355,Z 263.196,A -85,B 0,C 180,E1 -852.024,E2 -852.024} C_VEL
LIN {X 0,Y 753.324,Z 263.198,A -85,B 0,C 180,E1 -854.216,E2 -854.216} C_VEL
LIN {X 0,Y 753.391,Z 263.192,A -85,B 0,C 180,E1 -856.528,E2 -856.528} C_VEL
LIN {X 0,Y 753.415,Z 263.196,A -85,B 0,C 180,E1 -858.856,E2 -858.856} C_VEL
LIN {X 0,Y 753.372,Z 263.195,A -85,B 0,C 180,E1 -861.47,E2 -861.47} C_VEL
LIN {X 0,Y 753.377,Z 263.193,A -85,B 0,C 180,E1 -863.485,E2 -863.485} C_VEL
LIN {X 0,Y 753.395,Z 263.19,A -85,B 0,C 180,E1 -865.838,E2 -865.838} C_VEL
LIN {X 0,Y 753.367,Z 263.195,A -85,B 0,C 180,E1 -867.997,E2 -867.997} C_VEL
LIN {X 0,Y 753.379,Z 263.193,A -85,B 0,C 180,E1 -869.864,E2 -869.864} C_VEL
LIN {X 0,Y 753.389,Z 263.195,A -85,B 0,C 180,E1 -872.037,E2 -872.037} C_VEL
LIN {X 0,Y 753.42,Z 263.192,A -85,B 0,C 180,E1 -874.681,E2 -874.681} C_VEL
LIN {X 0,Y 753.412,Z 263.188,A -85,B 0,C 180,E1 -877.016,E2 -877.016} C_VEL
LIN {X 0,Y 753.412,Z 263.188,A -85,B 0,C 180,E1 -879.312,E2 -879.312} C_VEL
LIN {X 0,Y 753.391,Z 263.195,A -85,B 0,C 180,E1 -881.572,E2 -881.572} C_VEL
LIN {X 0,Y 753.398,Z 263.2,A -85,B 0,C 180,E1 -883.805,E2 -883.805} C_VEL
LIN {X 0,Y 753.396,Z 263.198,A -85,B 0,C 180,E1 -886.012,E2 -886.012} C_VEL
LIN {X 0,Y 753.41,Z 263.191,A -85,B 0,C 180,E1 -888.198,E2 -888.198} C_VEL
LIN {X 0,Y 753.439,Z 263.188,A -85,B 0,C 180,E1 -890.637,E2 -890.637} C_VEL
LIN {X 0,Y 753.451,Z 263.28,A -85,B 0,C 180,E1 -890.806,E2 -890.806} C_VEL
LIN {X 0,Y 753.589,Z 277.23,A -85,B 0,C 180,E1 -892.389,E2 -892.389} C_VEL
LIN {X 0,Y 753.519,Z 300.014,A -85,B 0,C 180,E1 -894.934,E2 -894.934} C_VEL
LIN {X 0,Y 753.473,Z 323.016,A -85,B 0,C 180,E1 -897.469,E2 -897.469} C_VEL
LIN {X 0,Y 753.454,Z 340.411,A -85,B 0,C 180,E1 -899.367,E2 -899.367} C_VEL
LIN {X 0,Y 753.635,Z 360.785,A -85,B 0,C 180,E1 -899.567,E2 -899.567} C_VEL
LIN {X 0,Y 753.575,Z 477.787,A -85,B 0,C 180,E1 -900.699,E2 -900.699} C_VEL
LIN {X 0,Y 753.578,Z 492.118,A -85,B 0,C 180,E1 -900.949,E2 -900.949} C_VEL
LIN {X 0,Y 753.514,Z 506.958,A -85,B 0,C 180,E1 -901.332,E2 -901.332} C_VEL
LIN {X 0,Y 753.494,Z 520.357,A -85,B 0,C 180,E1 -901.798,E2 -901.798} C_VEL
LIN {X 0,Y 753.487,Z 532.476,A -85,B 0,C 180,E1 -902.331,E2 -902.331} C_VEL
LIN {X 0,Y 753.449,Z 544.788,A -85,B 0,C 180,E1 -902.998,E2 -902.998} C_VEL
LIN {X 0,Y 753.418,Z 555.83,A -85,B 0,C 180,E1 -903.731,E2 -903.731} C_VEL
LIN {X 0,Y 753.416,Z 565.754,A -85,B 0,C 180,E1 -904.532,E2 -904.532} C_VEL
LIN {X 0,Y 753.388,Z 574.042,A -85,B 0,C 180,E1 -905.335,E2 -905.335} C_VEL
LIN {X 0,Y 753.362,Z 581.997,A -85,B 0,C 180,E1 -906.272,E2 -906.272} C_VEL
LIN {X 0,Y 753.373,Z 588.419,A -85,B 0,C 180,E1 -907.211,E2 -907.211} C_VEL
LIN {X 0,Y 753.343,Z 594.13,A -85,B 0,C 180,E1 -908.286,E2 -908.286} C_VEL
LIN {X 0,Y 753.348,Z 597.401,A -85,B 0,C 180,E1 -909.094,E2 -909.094} C_VEL
LIN {X 0,Y 753.32,Z 600.315,A -85,B 0,C 180,E1 -910.118,E2 -910.118} C_VEL
LIN {X 0,Y 752.645,Z 601.239,A -85,B 0,C 180,E1 -910.558,E2 -910.558} C_VEL
LIN {X 0,Y 749.757,Z 602.136,A -85,B 0,C 180,E1 -911.278,E2 -911.278} C_VEL
LIN {X 0,Y 747.332,Z 602.453,A -85,B 0,C 180,E1 -911.859,E2 -911.859} C_VEL
LIN {X 0,Y 746.312,Z 602.431,A -85,B 0,C 180,E1 -912.308,E2 -912.308} C_VEL
LIN {X 0,Y 746.24,Z 602.384,A -85,B 0,C 180,E1 -912.459,E2 -912.459} C_VEL
LIN {X 0,Y 746.236,Z 601.17,A -85,B 0,C 180,E1 -913.572,E2 -913.572} C_VEL
LIN {X 0,Y 746.255,Z 598.521,A -85,B 0,C 180,E1 -914.68,E2 -914.68} C_VEL
LIN {X 0,Y 746.259,Z 594.334,A -85,B 0,C 180,E1 -915.795,E2 -915.795} C_VEL
LIN {X 0,Y 746.258,Z 589.252,A -85,B 0,C 180,E1 -916.786,E2 -916.786} C_VEL
LIN {X 0,Y 746.275,Z 582.839,A -85,B 0,C 180,E1 -917.761,E2 -917.761} C_VEL
LIN {X 0,Y 746.33,Z 574.672,A -85,B 0,C 180,E1 -918.75,E2 -918.75} C_VEL
LIN {X 0,Y 746.343,Z 566.032,A -85,B 0,C 180,E1 -919.604,E2 -919.604} C_VEL
LIN {X 0,Y 746.398,Z 555.506,A -85,B 0,C 180,E1 -920.461,E2 -920.461} C_VEL
LIN {X 0,Y 746.416,Z 544.778,A -85,B 0,C 180,E1 -921.179,E2 -921.179} C_VEL
LIN {X 0,Y 746.46,Z 532.901,A -85,B 0,C 180,E1 -921.831,E2 -921.831} C_VEL
LIN {X 0,Y 746.483,Z 521.716,A -85,B 0,C 180,E1 -922.335,E2 -922.335} C_VEL
LIN {X 0,Y 746.539,Z 508.855,A -85,B 0,C 180,E1 -922.802,E2 -922.802} C_VEL
LIN {X 0,Y 746.598,Z 493.923,A -85,B 0,C 180,E1 -923.206,E2 -923.206} C_VEL
LIN {X 0,Y 746.631,Z 480.281,A -85,B 0,C 180,E1 -923.461,E2 -923.461} C_VEL
LIN {X 0,Y 746.645,Z 462.419,A -85,B 0,C 180,E1 -923.662,E2 -923.662} C_VEL
LIN {X 0,Y 746.605,Z 341.713,A -85,B 0,C 180,E1 -924.826,E2 -924.826} C_VEL
LIN {X 0,Y 746.409,Z 340.422,A -85,B 0,C 180,E1 -924.843,E2 -924.843} C_VEL
LIN {X 0,Y 746.467,Z 318.606,A -85,B 0,C 180,E1 -927.25,E2 -927.25} C_VEL
LIN {X 0,Y 746.52,Z 298.326,A -85,B 0,C 180,E1 -929.511,E2 -929.511} C_VEL
LIN {X 0,Y 746.651,Z 276.209,A -85,B 0,C 180,E1 -932.008,E2 -932.008} C_VEL
LIN {X 0,Y 746.643,Z 266.138,A -85,B 0,C 180,E1 -933.159,E2 -933.159} C_VEL
LIN {X 0,Y 746.384,Z 264.069,A -85,B 0,C 180,E1 -933.425,E2 -933.425} C_VEL
LIN {X 0,Y 746.362,Z 264.076,A -85,B 0,C 180,E1 -936.186,E2 -936.186} C_VEL
LIN {X 0,Y 746.359,Z 264.068,A -85,B 0,C 180,E1 -938.835,E2 -938.835} C_VEL
LIN {X 0,Y 746.378,Z 264.065,A -85,B 0,C 180,E1 -941.342,E2 -941.342} C_VEL
LIN {X 0,Y 746.34,Z 264.08,A -85,B 0,C 180,E1 -943.987,E2 -943.987} C_VEL
LIN {X 0,Y 746.336,Z 264.073,A -85,B 0,C 180,E1 -946.274,E2 -946.274} C_VEL
LIN {X 0,Y 746.331,Z 264.071,A -85,B 0,C 180,E1 -948.931,E2 -948.931} C_VEL
LIN {X 0,Y 746.352,Z 264.076,A -85,B 0,C 180,E1 -951.726,E2 -951.726} C_VEL
LIN {X 0,Y 746.351,Z 264.072,A -85,B 0,C 180,E1 -953.814,E2 -953.814} C_VEL
LIN {X 0,Y 746.329,Z 264.07,A -85,B 0,C 180,E1 -956.376,E2 -956.376} C_VEL
LIN {X 0,Y 746.339,Z 264.072,A -85,B 0,C 180,E1 -958.654,E2 -958.654} C_VEL
LIN {X 0,Y 746.367,Z 264.072,A -85,B 0,C 180,E1 -960.789,E2 -960.789} C_VEL
LIN {X 0,Y 746.395,Z 264.069,A -85,B 0,C 180,E1 -963.226,E2 -963.226} C_VEL
LIN {X 0,Y 746.346,Z 264.069,A -85,B 0,C 180,E1 -965.609,E2 -965.609} C_VEL
LIN {X 0,Y 746.346,Z 264.069,A -85,B 0,C 180,E1 -967.95,E2 -967.95} C_VEL
LIN {X 0,Y 746.352,Z 264.073,A -85,B 0,C 180,E1 -970.253,E2 -970.253} C_VEL
LIN {X 0,Y 746.38,Z 264.075,A -85,B 0,C 180,E1 -972.523,E2 -972.523} C_VEL
LIN {X 0,Y 746.413,Z 264.06,A -85,B 0,C 180,E1 -975.143,E2 -975.143} C_VEL
LIN {X 0,Y 746.374,Z 264.066,A -85,B 0,C 180,E1 -977.534,E2 -977.534} C_VEL
LIN {X 0,Y 746.396,Z 264.067,A -85,B 0,C 180,E1 -979.728,E2 -979.728} C_VEL
LIN {X 0,Y 746.394,Z 264.074,A -85,B 0,C 180,E1 -981.907,E2 -981.907} C_VEL
LIN {X 0,Y 746.392,Z 264.07,A -85,B 0,C 180,E1 -984.125,E2 -984.125} C_VEL
LIN {X 0,Y 746.437,Z 264.217,A -85,B 0,C 180,E1 -985.222,E2 -985.222} C_VEL
LIN {X 0,Y 746.366,Z 282.362,A -85,B 0,C 180,E1 -987.847,E2 -987.847} C_VEL
LIN {X 0,Y 746.378,Z 292.201,A -85,B 0,C 180,E1 -989.259,E2 -989.259} C_VEL
LIN {X 0,Y 746.732,Z 299.767,A -85,B 0,C 180,E1 -989.344,E2 -989.344} C_VEL
LIN {X 0,Y 746.617,Z 427.329,A -85,B 0,C 180,E1 -990.587,E2 -990.587} C_VEL
LIN {X 0,Y 746.619,Z 441.08,A -85,B 0,C 180,E1 -990.822,E2 -990.822} C_VEL
LIN {X 0,Y 746.539,Z 455.156,A -85,B 0,C 180,E1 -991.175,E2 -991.175} C_VEL
LIN {X 0,Y 746.501,Z 469.82,A -85,B 0,C 180,E1 -991.679,E2 -991.679} C_VEL
LIN {X 0,Y 746.476,Z 482.037,A -85,B 0,C 180,E1 -992.217,E2 -992.217} C_VEL
LIN {X 0,Y 746.427,Z 493.258,A -85,B 0,C 180,E1 -992.823,E2 -992.823} C_VEL
LIN {X 0,Y 746.357,Z 503.626,A -85,B 0,C 180,E1 -993.496,E2 -993.496} C_VEL
LIN {X 0,Y 746.353,Z 512.351,A -85,B 0,C 180,E1 -994.17,E2 -994.17} C_VEL
LIN {X 0,Y 746.316,Z 521.196,A -85,B 0,C 180,E1 -994.979,E2 -994.979} C_VEL
LIN {X 0,Y 746.304,Z 529.708,A -85,B 0,C 180,E1 -995.924,E2 -995.924} C_VEL
LIN {X 0,Y 746.288,Z 535.687,A -85,B 0,C 180,E1 -996.736,E2 -996.736} C_VEL
LIN {X 0,Y 746.287,Z 542.078,A -85,B 0,C 180,E1 -997.82,E2 -997.82} C_VEL
LIN {X 0,Y 746.264,Z 545.783,A -85,B 0,C 180,E1 -998.636,E2 -998.636} C_VEL
LIN {X 0,Y 746.252,Z 549.484,A -85,B 0,C 180,E1 -999.753,E2 -999.753} C_VEL
LIN {X 0,Y 746.225,Z 551.623,A -85,B 0,C 180,E1 -1000.819,E2 -1000.819} C_VEL
LIN {X 0,Y 746.243,Z 552.47,A -85,B 0,C 180,E1 -1001.916,E2 -1001.916} C_VEL
LIN {X 0,Y 746.254,Z 551.94,A -85,B 0,C 180,E1 -1003.017,E2 -1003.017} C_VEL
LIN {X 0,Y 746.233,Z 550.031,A -85,B 0,C 180,E1 -1004.124,E2 -1004.124} C_VEL
LIN {X 0,Y 746.269,Z 546.641,A -85,B 0,C 180,E1 -1005.235,E2 -1005.235} C_VEL
LIN {X 0,Y 746.261,Z 541.641,A -85,B 0,C 180,E1 -1006.353,E2 -1006.353} C_VEL
LIN {X 0,Y 746.274,Z 536.75,A -85,B 0,C 180,E1 -1007.195,E2 -1007.195} C_VEL
LIN {X 0,Y 746.313,Z 529.572,A -85,B 0,C 180,E1 -1008.182,E2 -1008.182} C_VEL
LIN {X 0,Y 746.327,Z 521.978,A -85,B 0,C 180,E1 -1009.033,E2 -1009.033} C_VEL
LIN {X 0,Y 746.344,Z 512.931,A -85,B 0,C 180,E1 -1009.872,E2 -1009.872} C_VEL
LIN {X 0,Y 746.402,Z 503.499,A -85,B 0,C 180,E1 -1010.602,E2 -1010.602} C_VEL
LIN {X 0,Y 746.418,Z 492.338,A -85,B 0,C 180,E1 -1011.322,E2 -1011.322} C_VEL
LIN {X 0,Y 746.473,Z 479.627,A -85,B 0,C 180,E1 -1011.99,E2 -1011.99} C_VEL
LIN {X 0,Y 746.503,Z 466.188,A -85,B 0,C 180,E1 -1012.551,E2 -1012.551} C_VEL
LIN {X 0,Y 746.583,Z 452.961,A -85,B 0,C 180,E1 -1012.976,E2 -1012.976} C_VEL
LIN {X 0,Y 746.594,Z 439.707,A -85,B 0,C 180,E1 -1013.296,E2 -1013.296} C_VEL
LIN {X 0,Y 746.602,Z 426.452,A -85,B 0,C 180,E1 -1013.515,E2 -1013.515} C_VEL
LIN {X 0,Y 746.617,Z 293.786,A -85,B 0,C 180,E1 -1014.806,E2 -1014.806} C_VEL
LIN {X 0,Y 746.354,Z 292.173,A -85,B 0,C 180,E1 -1014.835,E2 -1014.835} C_VEL
LIN {X 0,Y 746.386,Z 274.512,A -85,B 0,C 180,E1 -1017.375,E2 -1017.375} C_VEL
LIN {X 0,Y 746.363,Z 264.07,A -85,B 0,C 180,E1 -1018.9,E2 -1018.9} C_VEL
LIN {X 0,Y 746.315,Z 264.072,A -85,B 0,C 180,E1 -1021.343,E2 -1021.343} C_VEL
LIN {X 0,Y 746.32,Z 264.073,A -85,B 0,C 180,E1 -1023.621,E2 -1023.621} C_VEL
LIN {X 0,Y 746.34,Z 264.08,A -85,B 0,C 180,E1 -1026.244,E2 -1026.244} C_VEL
LIN {X 0,Y 746.346,Z 264.068,A -85,B 0,C 180,E1 -1028.835,E2 -1028.835} C_VEL
LIN {X 0,Y 746.358,Z 264.066,A -85,B 0,C 180,E1 -1031.341,E2 -1031.341} C_VEL
LIN {X 0,Y 746.335,Z 264.081,A -85,B 0,C 180,E1 -1033.985,E2 -1033.985} C_VEL
LIN {X 0,Y 746.343,Z 264.074,A -85,B 0,C 180,E1 -1036.271,E2 -1036.271} C_VEL
LIN {X 0,Y 746.335,Z 264.069,A -85,B 0,C 180,E1 -1038.932,E2 -1038.932} C_VEL
LIN {X 0,Y 746.345,Z 264.068,A -85,B 0,C 180,E1 -1041.162,E2 -1041.162} C_VEL
LIN {X 0,Y 746.339,Z 264.08,A -85,B 0,C 180,E1 -1043.812,E2 -1043.812} C_VEL
LIN {X 0,Y 746.339,Z 264.07,A -85,B 0,C 180,E1 -1046.377,E2 -1046.377} C_VEL
LIN {X 0,Y 746.318,Z 264.07,A -85,B 0,C 180,E1 -1048.652,E2 -1048.652} C_VEL
LIN {X 0,Y 746.337,Z 264.068,A -85,B 0,C 180,E1 -1050.789,E2 -1050.789} C_VEL
LIN {X 0,Y 746.342,Z 264.072,A -85,B 0,C 180,E1 -1053.225,E2 -1053.225} C_VEL
LIN {X 0,Y 746.377,Z 264.076,A -85,B 0,C 180,E1 -1055.611,E2 -1055.611} C_VEL
LIN {X 0,Y 746.34,Z 264.069,A -85,B 0,C 180,E1 -1058.292,E2 -1058.292} C_VEL
LIN {X 0,Y 746.333,Z 264.069,A -85,B 0,C 180,E1 -1060.253,E2 -1060.253} C_VEL
LIN {X 0,Y 746.341,Z 264.068,A -85,B 0,C 180,E1 -1062.523,E2 -1062.523} C_VEL
LIN {X 0,Y 746.332,Z 264.07,A -85,B 0,C 180,E1 -1064.765,E2 -1064.765} C_VEL
LIN {X 0,Y 746.384,Z 264.072,A -85,B 0,C 180,E1 -1067.535,E2 -1067.535} C_VEL
LIN {X 0,Y 746.37,Z 264.068,A -85,B 0,C 180,E1 -1069.729,E2 -1069.729} C_VEL
LIN {X 0,Y 746.369,Z 264.066,A -85,B 0,C 180,E1 -1071.908,E2 -1071.908} C_VEL
LIN {X 0,Y 746.336,Z 264.068,A -85,B 0,C 180,E1 -1074.144,E2 -1074.144} C_VEL
LIN {X 0,Y 746.312,Z 264.07,A -85,B 0,C 180,E1 -1076.233,E2 -1076.233} C_VEL
LIN {X 0,Y 746.344,Z 264.068,A -85,B 0,C 180,E1 -1078.387,E2 -1078.387} C_VEL
LIN {X 0,Y 746.345,Z 264.067,A -85,B 0,C 180,E1 -1080,E2 -1080} C_VEL
LIN {X 0,Y 746.349,Z 264.066,A -85,B 0,C 180,E1 -1082.151,E2 -1082.151} C_VEL
LIN {X 0,Y 746.388,Z 264.071,A -85,B 0,C 180,E1 -1084.845,E2 -1084.845} C_VEL
LIN {X 0,Y 746.396,Z 264.063,A -85,B 0,C 180,E1 -1087.549,E2 -1087.549} C_VEL
LIN {X 0,Y 746.344,Z 264.067,A -85,B 0,C 180,E1 -1089.807,E2 -1089.807} C_VEL
LIN {X 0,Y 746.35,Z 264.066,A -85,B 0,C 180,E1 -1091.916,E2 -1091.916} C_VEL
LIN {X 0,Y 746.318,Z 264.071,A -85,B 0,C 180,E1 -1094.124,E2 -1094.124} C_VEL
LIN {X 0,Y 746.355,Z 264.07,A -85,B 0,C 180,E1 -1096.353,E2 -1096.353} C_VEL
LIN {X 0,Y 746.382,Z 264.072,A -85,B 0,C 180,E1 -1098.607,E2 -1098.607} C_VEL
LIN {X 0,Y 746.358,Z 264.074,A -85,B 0,C 180,E1 -1100.893,E2 -1100.893} C_VEL
LIN {X 0,Y 746.375,Z 264.066,A -85,B 0,C 180,E1 -1103.213,E2 -1103.213} C_VEL
LIN {X 0,Y 746.359,Z 264.065,A -85,B 0,C 180,E1 -1105.723,E2 -1105.723} C_VEL
LIN {X 0,Y 746.36,Z 264.069,A -85,B 0,C 180,E1 -1108.099,E2 -1108.099} C_VEL
LIN {X 0,Y 746.34,Z 264.08,A -85,B 0,C 180,E1 -1110.451,E2 -1110.451} C_VEL
LIN {X 0,Y 746.361,Z 264.068,A -85,B 0,C 180,E1 -1112.978,E2 -1112.978} C_VEL
LIN {X 0,Y 746.342,Z 264.066,A -85,B 0,C 180,E1 -1115.268,E2 -1115.268} C_VEL
LIN {X 0,Y 746.34,Z 264.068,A -85,B 0,C 180,E1 -1117.592,E2 -1117.592} C_VEL
LIN {X 0,Y 746.362,Z 264.067,A -85,B 0,C 180,E1 -1119.69,E2 -1119.69} C_VEL
LIN {X 0,Y 746.351,Z 264.07,A -85,B 0,C 180,E1 -1121.784,E2 -1121.784} C_VEL
LIN {X 0,Y 746.342,Z 264.075,A -85,B 0,C 180,E1 -1123.987,E2 -1123.987} C_VEL
LIN {X 0,Y 746.358,Z 264.077,A -85,B 0,C 180,E1 -1126.272,E2 -1126.272} C_VEL
LIN {X 0,Y 746.383,Z 264.063,A -85,B 0,C 180,E1 -1128.937,E2 -1128.937} C_VEL
LIN {X 0,Y 746.357,Z 264.066,A -85,B 0,C 180,E1 -1131.164,E2 -1131.164} C_VEL
LIN {X 0,Y 746.344,Z 264.074,A -85,B 0,C 180,E1 -1133.756,E2 -1133.756} C_VEL
LIN {X 0,Y 746.354,Z 264.072,A -85,B 0,C 180,E1 -1136.38,E2 -1136.38} C_VEL
LIN {X 0,Y 746.346,Z 264.069,A -85,B 0,C 180,E1 -1138.653,E2 -1138.653} C_VEL
LIN {X 0,Y 746.357,Z 264.066,A -85,B 0,C 180,E1 -1140.792,E2 -1140.792} C_VEL
LIN {X 0,Y 746.349,Z 264.069,A -85,B 0,C 180,E1 -1143.228,E2 -1143.228} C_VEL
LIN {X 0,Y 746.364,Z 264.074,A -85,B 0,C 180,E1 -1145.613,E2 -1145.613} C_VEL
LIN {X 0,Y 746.385,Z 264.182,A -85,B 0,C 180,E1 -1146.771,E2 -1146.771} C_VEL
LIN {X 0,Y 746.825,Z 268.723,A -85,B 0,C 180,E1 -1147.248,E2 -1147.248} C_VEL
LIN {X 0,Y 746.746,Z 291.538,A -85,B 0,C 180,E1 -1149.551,E2 -1149.551} C_VEL
LIN {X 0,Y 746.612,Z 318.716,A -85,B 0,C 180,E1 -1152.249,E2 -1152.249} C_VEL
LIN {X 0,Y 746.536,Z 344.464,A -85,B 0,C 180,E1 -1154.771,E2 -1154.771} C_VEL
LIN {X 0,Y 746.467,Z 369.652,A -85,B 0,C 180,E1 -1157.196,E2 -1157.196} C_VEL
LIN {X 0,Y 746.747,Z 375.189,A -85,B 0,C 180,E1 -1157.255,E2 -1157.255} C_VEL
LIN {X 0,Y 746.613,Z 507.128,A -85,B 0,C 180,E1 -1158.536,E2 -1158.536} C_VEL
LIN {X 0,Y 746.609,Z 521.855,A -85,B 0,C 180,E1 -1158.793,E2 -1158.793} C_VEL
LIN {X 0,Y 746.566,Z 535.845,A -85,B 0,C 180,E1 -1159.152,E2 -1159.152} C_VEL
LIN {X 0,Y 746.489,Z 548.828,A -85,B 0,C 180,E1 -1159.595,E2 -1159.595} C_VEL
LIN {X 0,Y 746.448,Z 561.811,A -85,B 0,C 180,E1 -1160.16,E2 -1160.16} C_VEL
LIN {X 0,Y 746.42,Z 574.028,A -85,B 0,C 180,E1 -1160.822,E2 -1160.822} C_VEL
LIN {X 0,Y 746.367,Z 584.363,A -85,B 0,C 180,E1 -1161.501,E2 -1161.501} C_VEL
LIN {X 0,Y 746.354,Z 594.654,A -85,B 0,C 180,E1 -1162.316,E2 -1162.316} C_VEL
LIN {X 0,Y 746.33,Z 603.151,A -85,B 0,C 180,E1 -1163.129,E2 -1163.129} C_VEL
LIN {X 0,Y 746.304,Z 611.275,A -85,B 0,C 180,E1 -1164.076,E2 -1164.076} C_VEL
LIN {X 0,Y 746.305,Z 616.989,A -85,B 0,C 180,E1 -1164.886,E2 -1164.886} C_VEL
LIN {X 0,Y 746.243,Z 621.651,A -85,B 0,C 180,E1 -1165.695,E2 -1165.695} C_VEL
LIN {X 0,Y 746.255,Z 626.49,A -85,B 0,C 180,E1 -1166.773,E2 -1166.773} C_VEL
LIN {X 0,Y 746.224,Z 629.855,A -85,B 0,C 180,E1 -1167.85,E2 -1167.85} C_VEL
LIN {X 0,Y 746.251,Z 631.839,A -85,B 0,C 180,E1 -1168.926,E2 -1168.926} C_VEL
LIN {X 0,Y 746.24,Z 632.5,A -85,B 0,C 180,E1 -1170.001,E2 -1170.001} C_VEL
LIN {X 0,Y 746.251,Z 631.834,A -85,B 0,C 180,E1 -1171.077,E2 -1171.077} C_VEL
LIN {X 0,Y 746.224,Z 629.847,A -85,B 0,C 180,E1 -1172.153,E2 -1172.153} C_VEL
LIN {X 0,Y 746.256,Z 626.479,A -85,B 0,C 180,E1 -1173.23,E2 -1173.23} C_VEL
LIN {X 0,Y 746.243,Z 621.638,A -85,B 0,C 180,E1 -1174.308,E2 -1174.308} C_VEL
LIN {X 0,Y 746.305,Z 616.971,A -85,B 0,C 180,E1 -1175.117,E2 -1175.117} C_VEL
LIN {X 0,Y 746.306,Z 610.196,A -85,B 0,C 180,E1 -1176.062,E2 -1176.062} C_VEL
LIN {X 0,Y 746.307,Z 601.783,A -85,B 0,C 180,E1 -1177.009,E2 -1177.009} C_VEL
LIN {X 0,Y 746.351,Z 593.009,A -85,B 0,C 180,E1 -1177.822,E2 -1177.822} C_VEL
LIN {X 0,Y 746.361,Z 582.393,A -85,B 0,C 180,E1 -1178.637,E2 -1178.637} C_VEL
LIN {X 0,Y 746.45,Z 570.501,A -85,B 0,C 180,E1 -1179.385,E2 -1179.385} C_VEL
LIN {X 0,Y 746.49,Z 559.088,A -85,B 0,C 180,E1 -1179.97,E2 -1179.97} C_VEL
LIN {X 0,Y 746.496,Z 547.006,A -85,B 0,C 180,E1 -1180.476,E2 -1180.476} C_VEL
LIN {X 0,Y 746.579,Z 533.489,A -85,B 0,C 180,E1 -1180.919,E2 -1180.919} C_VEL
LIN {X 0,Y 746.61,Z 519.267,A -85,B 0,C 180,E1 -1181.261,E2 -1181.261} C_VEL
LIN {X 0,Y 746.639,Z 505.449,A -85,B 0,C 180,E1 -1181.483,E2 -1181.483} C_VEL
LIN {X 0,Y 746.639,Z 370.865,A -85,B 0,C 180,E1 -1182.789,E2 -1182.789} C_VEL
LIN {X 0,Y 746.449,Z 369.482,A -85,B 0,C 180,E1 -1182.808,E2 -1182.808} C_VEL
LIN {X 0,Y 746.541,Z 344.436,A -85,B 0,C 180,E1 -1185.232,E2 -1185.232} C_VEL
LIN {X 0,Y 746.634,Z 317.258,A -85,B 0,C 180,E1 -1187.894,E2 -1187.894} C_VEL
LIN {X 0,Y 746.72,Z 292.941,A -85,B 0,C 180,E1 -1190.309,E2 -1190.309} C_VEL
LIN {X 0,Y 746.826,Z 268.711,A -85,B 0,C 180,E1 -1192.753,E2 -1192.753} C_VEL
LIN {X 0,Y 746.368,Z 264.071,A -85,B 0,C 180,E1 -1193.251,E2 -1193.251} C_VEL
LIN {X 0,Y 746.392,Z 264.068,A -85,B 0,C 180,E1 -1195.723,E2 -1195.723} C_VEL
LIN {X 0,Y 746.381,Z 264.073,A -85,B 0,C 180,E1 -1198.097,E2 -1198.097} C_VEL
LIN {X 0,Y 746.347,Z 264.07,A -85,B 0,C 180,E1 -1200.451,E2 -1200.451} C_VEL
LIN {X 0,Y 746.355,Z 264.067,A -85,B 0,C 180,E1 -1202.979,E2 -1202.979} C_VEL
LIN {X 0,Y 746.325,Z 264.076,A -85,B 0,C 180,E1 -1205.262,E2 -1205.262} C_VEL
LIN {X 0,Y 746.358,Z 264.078,A -85,B 0,C 180,E1 -1207.591,E2 -1207.591} C_VEL
LIN {X 0,Y 746.332,Z 264.077,A -85,B 0,C 180,E1 -1209.683,E2 -1209.683} C_VEL
LIN {X 0,Y 746.344,Z 264.072,A -85,B 0,C 180,E1 -1211.786,E2 -1211.786} C_VEL
LIN {X 0,Y 746.315,Z 264.072,A -85,B 0,C 180,E1 -1213.99,E2 -1213.99} C_VEL
LIN {X 0,Y 746.332,Z 264.07,A -85,B 0,C 180,E1 -1216.275,E2 -1216.275} C_VEL
LIN {X 0,Y 746.366,Z 264.076,A -85,B 0,C 180,E1 -1218.934,E2 -1218.934} C_VEL
LIN {X 0,Y 746.364,Z 264.073,A -85,B 0,C 180,E1 -1221.164,E2 -1221.164} C_VEL
LIN {X 0,Y 746.344,Z 264.068,A -85,B 0,C 180,E1 -1223.816,E2 -1223.816} C_VEL
LIN {X 0,Y 746.353,Z 264.067,A -85,B 0,C 180,E1 -1225.73,E2 -1225.73} C_VEL
LIN {X 0,Y 746.35,Z 264.067,A -85,B 0,C 180,E1 -1227.66,E2 -1227.66} C_VEL
LIN {X 0,Y 746.357,Z 264.072,A -85,B 0,C 180,E1 -1230.172,E2 -1230.172} C_VEL
LIN {X 0,Y 746.355,Z 264.075,A -85,B 0,C 180,E1 -1232.622,E2 -1232.622} C_VEL
LIN {X 0,Y 746.343,Z 264.069,A -85,B 0,C 180,E1 -1235.018,E2 -1235.018} C_VEL
LIN {X 0,Y 746.352,Z 264.068,A -85,B 0,C 180,E1 -1237.37,E2 -1237.37} C_VEL
LIN {X 0,Y 746.394,Z 264.069,A -85,B 0,C 180,E1 -1239.792,E2 -1239.792} C_VEL
LIN {X 0,Y 746.376,Z 264.067,A -85,B 0,C 180,E1 -1242.524,E2 -1242.524} C_VEL
LIN {X 0,Y 746.37,Z 264.066,A -85,B 0,C 180,E1 -1245.156,E2 -1245.156} C_VEL
LIN {X 0,Y 746.379,Z 264.073,A -85,B 0,C 180,E1 -1247.535,E2 -1247.535} C_VEL
LIN {X 0,Y 746.392,Z 264.075,A -85,B 0,C 180,E1 -1249.729,E2 -1249.729} C_VEL
LIN {X 0,Y 746.431,Z 264.196,A -85,B 0,C 180,E1 -1250.701,E2 -1250.701} C_VEL
LIN {X 0,Y 746.663,Z 269.945,A -85,B 0,C 180,E1 -1251.367,E2 -1251.367} C_VEL
LIN {X 0,Y 746.589,Z 290.362,A -85,B 0,C 180,E1 -1253.684,E2 -1253.684} C_VEL
LIN {X 0,Y 746.493,Z 314.353,A -85,B 0,C 180,E1 -1256.369,E2 -1256.369} C_VEL
LIN {X 0,Y 746.444,Z 338.705,A -85,B 0,C 180,E1 -1259.059,E2 -1259.059} C_VEL
LIN {X 0,Y 746.423,Z 340.391,A -85,B 0,C 180,E1 -1259.244,E2 -1259.244} C_VEL
LIN {X 0,Y 746.764,Z 346.365,A -85,B 0,C 180,E1 -1259.311,E2 -1259.311} C_VEL
LIN {X 0,Y 746.613,Z 477.476,A -85,B 0,C 180,E1 -1260.588,E2 -1260.588} C_VEL
LIN {X 0,Y 746.615,Z 491.135,A -85,B 0,C 180,E1 -1260.823,E2 -1260.823} C_VEL
LIN {X 0,Y 746.534,Z 505.193,A -85,B 0,C 180,E1 -1261.176,E2 -1261.176} C_VEL
LIN {X 0,Y 746.499,Z 518.115,A -85,B 0,C 180,E1 -1261.613,E2 -1261.613} C_VEL
LIN {X 0,Y 746.458,Z 530.668,A -85,B 0,C 180,E1 -1262.151,E2 -1262.151} C_VEL
LIN {X 0,Y 746.434,Z 542.154,A -85,B 0,C 180,E1 -1262.757,E2 -1262.757} C_VEL
LIN {X 0,Y 746.359,Z 553.674,A -85,B 0,C 180,E1 -1263.497,E2 -1263.497} C_VEL
LIN {X 0,Y 746.361,Z 564.007,A -85,B 0,C 180,E1 -1264.306,E2 -1264.306} C_VEL
LIN {X 0,Y 746.325,Z 572.571,A -85,B 0,C 180,E1 -1265.115,E2 -1265.115} C_VEL
LIN {X 0,Y 746.307,Z 580.818,A -85,B 0,C 180,E1 -1266.061,E2 -1266.061} C_VEL
LIN {X 0,Y 746.279,Z 587.477,A -85,B 0,C 180,E1 -1267.008,E2 -1267.008} C_VEL
LIN {X 0,Y 746.243,Z 593.415,A -85,B 0,C 180,E1 -1268.094,E2 -1268.094} C_VEL
LIN {X 0,Y 746.259,Z 597.78,A -85,B 0,C 180,E1 -1269.182,E2 -1269.182} C_VEL
LIN {X 0,Y 746.227,Z 600.694,A -85,B 0,C 180,E1 -1270.273,E2 -1270.273} C_VEL
LIN {X 0,Y 746.228,Z 602.218,A -85,B 0,C 180,E1 -1271.368,E2 -1271.368} C_VEL
LIN {X 0,Y 746.24,Z 602.384,A -85,B 0,C 180,E1 -1272.459,E2 -1272.459} C_VEL
LIN {X 0,Y 745.59,Z 602.137,A -85,B 0,C 180,E1 -1272.909,E2 -1272.909} C_VEL
LIN {X 0,Y 742.701,Z 601.088,A -85,B 0,C 180,E1 -1273.634,E2 -1273.634} C_VEL
LIN {X 0,Y 740.267,Z 599.858,A -85,B 0,C 180,E1 -1274.213,E2 -1274.213} C_VEL
LIN {X 0,Y 739.251,Z 598.669,A -85,B 0,C 180,E1 -1274.656,E2 -1274.656} C_VEL
LIN {X 0,Y 739.187,Z 598.194,A -85,B 0,C 180,E1 -1274.806,E2 -1274.806} C_VEL
LIN {X 0,Y 739.168,Z 593.793,A -85,B 0,C 180,E1 -1275.951,E2 -1275.951} C_VEL
LIN {X 0,Y 739.177,Z 589.167,A -85,B 0,C 180,E1 -1276.847,E2 -1276.847} C_VEL
LIN {X 0,Y 739.206,Z 583.004,A -85,B 0,C 180,E1 -1277.794,E2 -1277.794} C_VEL
LIN {X 0,Y 739.25,Z 574.869,A -85,B 0,C 180,E1 -1278.793,E2 -1278.793} C_VEL
LIN {X 0,Y 739.289,Z 566.27,A -85,B 0,C 180,E1 -1279.654,E2 -1279.654} C_VEL
LIN {X 0,Y 739.36,Z 555.797,A -85,B 0,C 180,E1 -1280.519,E2 -1280.519} C_VEL
LIN {X 0,Y 739.387,Z 545.139,A -85,B 0,C 180,E1 -1281.245,E2 -1281.245} C_VEL
LIN {X 0,Y 739.45,Z 532.453,A -85,B 0,C 180,E1 -1281.946,E2 -1281.946} C_VEL
LIN {X 0,Y 739.478,Z 520.438,A -85,B 0,C 180,E1 -1282.485,E2 -1282.485} C_VEL
LIN {X 0,Y 739.595,Z 506.93,A -85,B 0,C 180,E1 -1282.964,E2 -1282.964} C_VEL
LIN {X 0,Y 739.642,Z 492.068,A -85,B 0,C 180,E1 -1283.354,E2 -1283.354} C_VEL
LIN {X 0,Y 739.68,Z 479.308,A -85,B 0,C 180,E1 -1283.584,E2 -1283.584} C_VEL
LIN {X 0,Y 739.679,Z 459.021,A -85,B 0,C 180,E1 -1283.806,E2 -1283.806} C_VEL
LIN {X 0,Y 739.64,Z 342.373,A -85,B 0,C 180,E1 -1284.942,E2 -1284.942} C_VEL
LIN {X 0,Y 739.36,Z 340.339,A -85,B 0,C 180,E1 -1284.976,E2 -1284.976} C_VEL
LIN {X 0,Y 739.475,Z 319.31,A -85,B 0,C 180,E1 -1287.318,E2 -1287.318} C_VEL
LIN {X 0,Y 739.554,Z 298.502,A -85,B 0,C 180,E1 -1289.661,E2 -1289.661} C_VEL
LIN {X 0,Y 739.697,Z 276.373,A -85,B 0,C 180,E1 -1292.185,E2 -1292.185} C_VEL
LIN {X 0,Y 739.59,Z 266.58,A -85,B 0,C 180,E1 -1293.319,E2 -1293.319} C_VEL
LIN {X 0,Y 739.343,Z 264.947,A -85,B 0,C 180,E1 -1293.536,E2 -1293.536} C_VEL
LIN {X 0,Y 739.31,Z 264.95,A -85,B 0,C 180,E1 -1295.973,E2 -1295.973} C_VEL
LIN {X 0,Y 739.334,Z 264.952,A -85,B 0,C 180,E1 -1298.154,E2 -1298.154} C_VEL
LIN {X 0,Y 739.309,Z 264.946,A -85,B 0,C 180,E1 -1300.823,E2 -1300.823} C_VEL
LIN {X 0,Y 739.284,Z 264.948,A -85,B 0,C 180,E1 -1303.151,E2 -1303.151} C_VEL
LIN {X 0,Y 739.297,Z 264.951,A -85,B 0,C 180,E1 -1305.483,E2 -1305.483} C_VEL
LIN {X 0,Y 739.287,Z 264.959,A -85,B 0,C 180,E1 -1307.724,E2 -1307.724} C_VEL
LIN {X 0,Y 739.261,Z 264.954,A -85,B 0,C 180,E1 -1310.127,E2 -1310.127} C_VEL
LIN {X 0,Y 739.284,Z 264.952,A -85,B 0,C 180,E1 -1311.985,E2 -1311.985} C_VEL
LIN {X 0,Y 739.295,Z 264.949,A -85,B 0,C 180,E1 -1314.025,E2 -1314.025} C_VEL
LIN {X 0,Y 739.29,Z 264.948,A -85,B 0,C 180,E1 -1316.487,E2 -1316.487} C_VEL
LIN {X 0,Y 739.299,Z 264.948,A -85,B 0,C 180,E1 -1318.593,E2 -1318.593} C_VEL
LIN {X 0,Y 739.327,Z 264.954,A -85,B 0,C 180,E1 -1321.106,E2 -1321.106} C_VEL
LIN {X 0,Y 739.317,Z 264.946,A -85,B 0,C 180,E1 -1323.557,E2 -1323.557} C_VEL
LIN {X 0,Y 739.291,Z 264.948,A -85,B 0,C 180,E1 -1325.957,E2 -1325.957} C_VEL
LIN {X 0,Y 739.34,Z 264.946,A -85,B 0,C 180,E1 -1328.315,E2 -1328.315} C_VEL
LIN {X 0,Y 739.33,Z 264.953,A -85,B 0,C 180,E1 -1330.634,E2 -1330.634} C_VEL
LIN {X 0,Y 739.371,Z 264.938,A -85,B 0,C 180,E1 -1333.102,E2 -1333.102} C_VEL
LIN {X 0,Y 739.315,Z 264.947,A -85,B 0,C 180,E1 -1335.738,E2 -1335.738} C_VEL
LIN {X 0,Y 739.339,Z 264.949,A -85,B 0,C 180,E1 -1337.969,E2 -1337.969} C_VEL
LIN {X 0,Y 739.334,Z 264.951,A -85,B 0,C 180,E1 -1340.18,E2 -1340.18} C_VEL
LIN {X 0,Y 739.329,Z 264.947,A -85,B 0,C 180,E1 -1342.377,E2 -1342.377} C_VEL
LIN {X 0,Y 739.307,Z 264.948,A -85,B 0,C 180,E1 -1344.562,E2 -1344.562} C_VEL
LIN {X 0,Y 739.383,Z 265.03,A -85,B 0,C 180,E1 -1345.176,E2 -1345.176} C_VEL
LIN {X 0,Y 739.335,Z 283.17,A -85,B 0,C 180,E1 -1347.827,E2 -1347.827} C_VEL
LIN {X 0,Y 739.343,Z 292.187,A -85,B 0,C 180,E1 -1349.134,E2 -1349.134} C_VEL
LIN {X 0,Y 739.807,Z 297.627,A -85,B 0,C 180,E1 -1349.202,E2 -1349.202} C_VEL
LIN {X 0,Y 739.66,Z 426.955,A -85,B 0,C 180,E1 -1350.473,E2 -1350.473} C_VEL
LIN {X 0,Y 739.663,Z 439.979,A -85,B 0,C 180,E1 -1350.694,E2 -1350.694} C_VEL
LIN {X 0,Y 739.602,Z 453.185,A -85,B 0,C 180,E1 -1351.016,E2 -1351.016} C_VEL
LIN {X 0,Y 739.503,Z 465.742,A -85,B 0,C 180,E1 -1351.423,E2 -1351.423} C_VEL
LIN {X 0,Y 739.47,Z 478.836,A -85,B 0,C 180,E1 -1351.966,E2 -1351.966} C_VEL
LIN {X 0,Y 739.409,Z 491.762,A -85,B 0,C 180,E1 -1352.646,E2 -1352.646} C_VEL
LIN {X 0,Y 739.347,Z 501.409,A -85,B 0,C 180,E1 -1353.257,E2 -1353.257} C_VEL
LIN {X 0,Y 739.33,Z 510.484,A -85,B 0,C 180,E1 -1353.937,E2 -1353.937} C_VEL
LIN {X 0,Y 739.237,Z 519.628,A -85,B 0,C 180,E1 -1354.754,E2 -1354.754} C_VEL
LIN {X 0,Y 739.197,Z 527.268,A -85,B 0,C 180,E1 -1355.571,E2 -1355.571} C_VEL
LIN {X 0,Y 739.215,Z 532.689,A -85,B 0,C 180,E1 -1356.254,E2 -1356.254} C_VEL
LIN {X 0,Y 739.183,Z 538.161,A -85,B 0,C 180,E1 -1357.075,E2 -1357.075} C_VEL
LIN {X 0,Y 739.187,Z 542.674,A -85,B 0,C 180,E1 -1357.896,E2 -1357.896} C_VEL
LIN {X 0,Y 739.183,Z 546.237,A -85,B 0,C 180,E1 -1358.719,E2 -1358.719} C_VEL
LIN {X 0,Y 739.146,Z 549.721,A -85,B 0,C 180,E1 -1359.82,E2 -1359.82} C_VEL
LIN {X 0,Y 739.132,Z 551.781,A -85,B 0,C 180,E1 -1360.924,E2 -1360.924} C_VEL
LIN {X 0,Y 739.143,Z 552.466,A -85,B 0,C 180,E1 -1362.032,E2 -1362.032} C_VEL
LIN {X 0,Y 739.183,Z 552.332,A -85,B 0,C 180,E1 -1362.587,E2 -1362.587} C_VEL
LIN {X 0,Y 739.131,Z 550.943,A -85,B 0,C 180,E1 -1363.703,E2 -1363.703} C_VEL
LIN {X 0,Y 739.145,Z 549.742,A -85,B 0,C 180,E1 -1364.262,E2 -1364.262} C_VEL
LIN {X 0,Y 739.18,Z 546.183,A -85,B 0,C 180,E1 -1365.385,E2 -1365.385} C_VEL
LIN {X 0,Y 739.181,Z 541.021,A -85,B 0,C 180,E1 -1366.514,E2 -1366.514} C_VEL
LIN {X 0,Y 739.189,Z 535.952,A -85,B 0,C 180,E1 -1367.365,E2 -1367.365} C_VEL
LIN {X 0,Y 739.24,Z 529.748,A -85,B 0,C 180,E1 -1368.219,E2 -1368.219} C_VEL
LIN {X 0,Y 739.266,Z 522.188,A -85,B 0,C 180,E1 -1369.078,E2 -1369.078} C_VEL
LIN {X 0,Y 739.289,Z 514.691,A -85,B 0,C 180,E1 -1369.797,E2 -1369.797} C_VEL
LIN {X 0,Y 739.333,Z 504.793,A -85,B 0,C 180,E1 -1370.591,E2 -1370.591} C_VEL
LIN {X 0,Y 739.384,Z 495.105,A -85,B 0,C 180,E1 -1371.243,E2 -1371.243} C_VEL
LIN {X 0,Y 739.459,Z 483.699,A -85,B 0,C 180,E1 -1371.883,E2 -1371.883} C_VEL
LIN {X 0,Y 739.511,Z 472.288,A -85,B 0,C 180,E1 -1372.408,E2 -1372.408} C_VEL
LIN {X 0,Y 739.556,Z 460.507,A -85,B 0,C 180,E1 -1372.848,E2 -1372.848} C_VEL
LIN {X 0,Y 739.606,Z 447.24,A -85,B 0,C 180,E1 -1373.234,E2 -1373.234} C_VEL
LIN {X 0,Y 739.657,Z 431.954,A -85,B 0,C 180,E1 -1373.546,E2 -1373.546} C_VEL
LIN {X 0,Y 739.654,Z 414.891,A -85,B 0,C 180,E1 -1373.749,E2 -1373.749} C_VEL
LIN {X 0,Y 739.799,Z 295.235,A -85,B 0,C 180,E1 -1374.912,E2 -1374.912} C_VEL
LIN {X 0,Y 739.297,Z 292.216,A -85,B 0,C 180,E1 -1374.953,E2 -1374.953} C_VEL
LIN {X 0,Y 739.345,Z 274.649,A -85,B 0,C 180,E1 -1377.504,E2 -1377.504} C_VEL
LIN {X 0,Y 739.338,Z 264.945,A -85,B 0,C 180,E1 -1378.944,E2 -1378.944} C_VEL
LIN {X 0,Y 739.275,Z 264.95,A -85,B 0,C 180,E1 -1381.49,E2 -1381.49} C_VEL
LIN {X 0,Y 739.302,Z 264.953,A -85,B 0,C 180,E1 -1383.984,E2 -1383.984} C_VEL
LIN {X 0,Y 739.285,Z 264.951,A -85,B 0,C 180,E1 -1386.646,E2 -1386.646} C_VEL
LIN {X 0,Y 739.309,Z 264.944,A -85,B 0,C 180,E1 -1389.023,E2 -1389.023} C_VEL
LIN {X 0,Y 739.309,Z 264.947,A -85,B 0,C 180,E1 -1391.542,E2 -1391.542} C_VEL
LIN {X 0,Y 739.305,Z 264.956,A -85,B 0,C 180,E1 -1393.941,E2 -1393.941} C_VEL
LIN {X 0,Y 739.297,Z 264.953,A -85,B 0,C 180,E1 -1396.24,E2 -1396.24} C_VEL
LIN {X 0,Y 739.336,Z 264.944,A -85,B 0,C 180,E1 -1398.457,E2 -1398.457} C_VEL
LIN {X 0,Y 739.316,Z 264.945,A -85,B 0,C 180,E1 -1401.296,E2 -1401.296} C_VEL
LIN {X 0,Y 739.283,Z 264.955,A -85,B 0,C 180,E1 -1403.64,E2 -1403.64} C_VEL
LIN {X 0,Y 739.307,Z 264.952,A -85,B 0,C 180,E1 -1406.014,E2 -1406.014} C_VEL
LIN {X 0,Y 739.283,Z 264.947,A -85,B 0,C 180,E1 -1408.594,E2 -1408.594} C_VEL
LIN {X 0,Y 739.296,Z 264.948,A -85,B 0,C 180,E1 -1411.105,E2 -1411.105} C_VEL
LIN {X 0,Y 739.285,Z 264.957,A -85,B 0,C 180,E1 -1413.557,E2 -1413.557} C_VEL
LIN {X 0,Y 739.303,Z 264.949,A -85,B 0,C 180,E1 -1415.958,E2 -1415.958} C_VEL
LIN {X 0,Y 739.303,Z 264.945,A -85,B 0,C 180,E1 -1418.315,E2 -1418.315} C_VEL
LIN {X 0,Y 739.301,Z 264.944,A -85,B 0,C 180,E1 -1420.634,E2 -1420.634} C_VEL
LIN {X 0,Y 739.315,Z 264.949,A -85,B 0,C 180,E1 -1423.109,E2 -1423.109} C_VEL
LIN {X 0,Y 739.29,Z 264.951,A -85,B 0,C 180,E1 -1425.739,E2 -1425.739} C_VEL
LIN {X 0,Y 739.321,Z 264.944,A -85,B 0,C 180,E1 -1427.97,E2 -1427.97} C_VEL
LIN {X 0,Y 739.303,Z 264.944,A -85,B 0,C 180,E1 -1430.181,E2 -1430.181} C_VEL
LIN {X 0,Y 739.357,Z 264.943,A -85,B 0,C 180,E1 -1432.926,E2 -1432.926} C_VEL
LIN {X 0,Y 739.377,Z 264.938,A -85,B 0,C 180,E1 -1435.654,E2 -1435.654} C_VEL
LIN {X 0,Y 739.32,Z 264.943,A -85,B 0,C 180,E1 -1438.371,E2 -1438.371} C_VEL
LIN {X 0,Y 739.281,Z 264.95,A -85,B 0,C 180,E1 -1440.543,E2 -1440.543} C_VEL
LIN {X 0,Y 739.318,Z 264.942,A -85,B 0,C 180,E1 -1442.172,E2 -1442.172} C_VEL
LIN {X 0,Y 739.36,Z 264.947,A -85,B 0,C 180,E1 -1444.891,E2 -1444.891} C_VEL
LIN {X 0,Y 739.358,Z 264.938,A -85,B 0,C 180,E1 -1447.622,E2 -1447.622} C_VEL
LIN {X 0,Y 739.324,Z 264.942,A -85,B 0,C 180,E1 -1449.847,E2 -1449.847} C_VEL
LIN {X 0,Y 739.308,Z 264.943,A -85,B 0,C 180,E1 -1452.031,E2 -1452.031} C_VEL
LIN {X 0,Y 739.352,Z 264.951,A -85,B 0,C 180,E1 -1454.821,E2 -1454.821} C_VEL
LIN {X 0,Y 739.339,Z 264.945,A -85,B 0,C 180,E1 -1457.079,E2 -1457.079} C_VEL
LIN {X 0,Y 739.312,Z 264.945,A -85,B 0,C 180,E1 -1459.366,E2 -1459.366} C_VEL
LIN {X 0,Y 739.293,Z 264.945,A -85,B 0,C 180,E1 -1461.803,E2 -1461.803} C_VEL
LIN {X 0,Y 739.282,Z 264.949,A -85,B 0,C 180,E1 -1464.042,E2 -1464.042} C_VEL
LIN {X 0,Y 739.305,Z 264.954,A -85,B 0,C 180,E1 -1466.442,E2 -1466.442} C_VEL
LIN {X 0,Y 739.328,Z 264.947,A -85,B 0,C 180,E1 -1468.893,E2 -1468.893} C_VEL
LIN {X 0,Y 739.296,Z 264.945,A -85,B 0,C 180,E1 -1471.497,E2 -1471.497} C_VEL
LIN {X 0,Y 739.329,Z 264.941,A -85,B 0,C 180,E1 -1473.521,E2 -1473.521} C_VEL
LIN {X 0,Y 739.3,Z 264.947,A -85,B 0,C 180,E1 -1475.974,E2 -1475.974} C_VEL
LIN {X 0,Y 739.326,Z 264.95,A -85,B 0,C 180,E1 -1478.158,E2 -1478.158} C_VEL
LIN {X 0,Y 739.33,Z 264.944,A -85,B 0,C 180,E1 -1480.822,E2 -1480.822} C_VEL
LIN {X 0,Y 739.307,Z 264.944,A -85,B 0,C 180,E1 -1483.156,E2 -1483.156} C_VEL
LIN {X 0,Y 739.315,Z 264.944,A -85,B 0,C 180,E1 -1485.488,E2 -1485.488} C_VEL
LIN {X 0,Y 739.297,Z 264.949,A -85,B 0,C 180,E1 -1487.728,E2 -1487.728} C_VEL
LIN {X 0,Y 739.328,Z 264.954,A -85,B 0,C 180,E1 -1490.121,E2 -1490.121} C_VEL
LIN {X 0,Y 739.315,Z 264.945,A -85,B 0,C 180,E1 -1492.734,E2 -1492.734} C_VEL
LIN {X 0,Y 739.326,Z 264.944,A -85,B 0,C 180,E1 -1495.36,E2 -1495.36} C_VEL
LIN {X 0,Y 739.312,Z 264.948,A -85,B 0,C 180,E1 -1497.481,E2 -1497.481} C_VEL
LIN {X 0,Y 739.311,Z 264.956,A -85,B 0,C 180,E1 -1499.861,E2 -1499.861} C_VEL
LIN {X 0,Y 739.311,Z 264.948,A -85,B 0,C 180,E1 -1502.341,E2 -1502.341} C_VEL
LIN {X 0,Y 739.313,Z 264.944,A -85,B 0,C 180,E1 -1504.766,E2 -1504.766} C_VEL
LIN {X 0,Y 739.342,Z 264.986,A -85,B 0,C 180,E1 -1506.641,E2 -1506.641} C_VEL
LIN {X 0,Y 739.937,Z 270.04,A -85,B 0,C 180,E1 -1507.164,E2 -1507.164} C_VEL
LIN {X 0,Y 739.844,Z 293.989,A -85,B 0,C 180,E1 -1509.6,E2 -1509.6} C_VEL
LIN {X 0,Y 739.629,Z 321.577,A -85,B 0,C 180,E1 -1512.361,E2 -1512.361} C_VEL
LIN {X 0,Y 739.526,Z 347.153,A -85,B 0,C 180,E1 -1514.887,E2 -1514.887} C_VEL
LIN {X 0,Y 739.434,Z 369.421,A -85,B 0,C 180,E1 -1517.062,E2 -1517.062} C_VEL
LIN {X 0,Y 739.838,Z 374.816,A -85,B 0,C 180,E1 -1517.13,E2 -1517.13} C_VEL
LIN {X 0,Y 739.679,Z 507.127,A -85,B 0,C 180,E1 -1518.427,E2 -1518.427} C_VEL
LIN {X 0,Y 739.67,Z 521.094,A -85,B 0,C 180,E1 -1518.669,E2 -1518.669} C_VEL
LIN {X 0,Y 739.602,Z 534.718,A -85,B 0,C 180,E1 -1519.014,E2 -1519.014} C_VEL
LIN {X 0,Y 739.517,Z 547.072,A -85,B 0,C 180,E1 -1519.427,E2 -1519.427} C_VEL
LIN {X 0,Y 739.49,Z 560,A -85,B 0,C 180,E1 -1519.979,E2 -1519.979} C_VEL
LIN {X 0,Y 739.424,Z 571.826,A -85,B 0,C 180,E1 -1520.603,E2 -1520.603} C_VEL
LIN {X 0,Y 739.325,Z 582.431,A -85,B 0,C 180,E1 -1521.283,E2 -1521.283} C_VEL
LIN {X 0,Y 739.287,Z 593.041,A -85,B 0,C 180,E1 -1522.105,E2 -1522.105} C_VEL
LIN {X 0,Y 739.255,Z 601.809,A -85,B 0,C 180,E1 -1522.926,E2 -1522.926} C_VEL
LIN {X 0,Y 739.237,Z 610.218,A -85,B 0,C 180,E1 -1523.882,E2 -1523.882} C_VEL
LIN {X 0,Y 739.217,Z 616.988,A -85,B 0,C 180,E1 -1524.837,E2 -1524.837} C_VEL
LIN {X 0,Y 739.149,Z 621.651,A -85,B 0,C 180,E1 -1525.654,E2 -1525.654} C_VEL
LIN {X 0,Y 739.159,Z 625.435,A -85,B 0,C 180,E1 -1526.47,E2 -1526.47} C_VEL
LIN {X 0,Y 739.166,Z 628.351,A -85,B 0,C 180,E1 -1527.286,E2 -1527.286} C_VEL
LIN {X 0,Y 739.138,Z 631.015,A -85,B 0,C 180,E1 -1528.372,E2 -1528.372} C_VEL
LIN {X 0,Y 739.141,Z 632.335,A -85,B 0,C 180,E1 -1529.458,E2 -1529.458} C_VEL
LIN {X 0,Y 739.141,Z 632.333,A -85,B 0,C 180,E1 -1530.544,E2 -1530.544} C_VEL
LIN {X 0,Y 739.138,Z 631.008,A -85,B 0,C 180,E1 -1531.63,E2 -1531.63} C_VEL
LIN {X 0,Y 739.166,Z 628.341,A -85,B 0,C 180,E1 -1532.717,E2 -1532.717} C_VEL
LIN {X 0,Y 739.22,Z 624.252,A -85,B 0,C 180,E1 -1533.804,E2 -1533.804} C_VEL
LIN {X 0,Y 739.213,Z 618.617,A -85,B 0,C 180,E1 -1534.893,E2 -1534.893} C_VEL
LIN {X 0,Y 739.189,Z 612.972,A -85,B 0,C 180,E1 -1535.752,E2 -1535.752} C_VEL
LIN {X 0,Y 739.251,Z 605.6,A -85,B 0,C 180,E1 -1536.667,E2 -1536.667} C_VEL
LIN {X 0,Y 739.294,Z 596.117,A -85,B 0,C 180,E1 -1537.624,E2 -1537.624} C_VEL
LIN {X 0,Y 739.323,Z 586.19,A -85,B 0,C 180,E1 -1538.446,E2 -1538.446} C_VEL
LIN {X 0,Y 739.377,Z 575.138,A -85,B 0,C 180,E1 -1539.2,E2 -1539.2} C_VEL
LIN {X 0,Y 739.433,Z 562.876,A -85,B 0,C 180,E1 -1539.882,E2 -1539.882} C_VEL
LIN {X 0,Y 739.489,Z 550.505,A -85,B 0,C 180,E1 -1540.438,E2 -1540.438} C_VEL
LIN {X 0,Y 739.569,Z 536.881,A -85,B 0,C 180,E1 -1540.92,E2 -1540.92} C_VEL
LIN {X 0,Y 739.616,Z 522.499,A -85,B 0,C 180,E1 -1541.3,E2 -1541.3} C_VEL
LIN {X 0,Y 739.657,Z 508.115,A -85,B 0,C 180,E1 -1541.558,E2 -1541.558} C_VEL
LIN {X 0,Y 739.798,Z 413.653,A -85,B 0,C 180,E1 -1542.492,E2 -1542.492} C_VEL
LIN {X 0,Y 739.663,Z 371.103,A -85,B 0,C 180,E1 -1542.909,E2 -1542.909} C_VEL
LIN {X 0,Y 739.44,Z 369.482,A -85,B 0,C 180,E1 -1542.932,E2 -1542.932} C_VEL
LIN {X 0,Y 739.544,Z 344.436,A -85,B 0,C 180,E1 -1545.38,E2 -1545.38} C_VEL
LIN {X 0,Y 739.665,Z 318.688,A -85,B 0,C 180,E1 -1547.926,E2 -1547.926} C_VEL
LIN {X 0,Y 739.793,Z 294.109,A -85,B 0,C 180,E1 -1550.39,E2 -1550.39} C_VEL
LIN {X 0,Y 739.963,Z 271.477,A -85,B 0,C 180,E1 -1552.691,E2 -1552.691} C_VEL
LIN {X 0,Y 739.525,Z 265.959,A -85,B 0,C 180,E1 -1553.257,E2 -1553.257} C_VEL
LIN {X 0,Y 739.327,Z 264.949,A -85,B 0,C 180,E1 -1553.38,E2 -1553.38} C_VEL
LIN {X 0,Y 739.331,Z 264.951,A -85,B 0,C 180,E1 -1555.838,E2 -1555.838} C_VEL
LIN {X 0,Y 739.316,Z 264.95,A -85,B 0,C 180,E1 -1558.276,E2 -1558.276} C_VEL
LIN {X 0,Y 739.304,Z 264.945,A -85,B 0,C 180,E1 -1560.773,E2 -1560.773} C_VEL
LIN {X 0,Y 739.324,Z 264.951,A -85,B 0,C 180,E1 -1563.517,E2 -1563.517} C_VEL
LIN {X 0,Y 739.298,Z 264.951,A -85,B 0,C 180,E1 -1565.975,E2 -1565.975} C_VEL
LIN {X 0,Y 739.314,Z 264.946,A -85,B 0,C 180,E1 -1568.153,E2 -1568.153} C_VEL
LIN {X 0,Y 739.303,Z 264.948,A -85,B 0,C 180,E1 -1570.825,E2 -1570.825} C_VEL
LIN {X 0,Y 739.284,Z 264.957,A -85,B 0,C 180,E1 -1573.152,E2 -1573.152} C_VEL
LIN {X 0,Y 739.302,Z 264.952,A -85,B 0,C 180,E1 -1575.484,E2 -1575.484} C_VEL
LIN {X 0,Y 739.276,Z 264.95,A -85,B 0,C 180,E1 -1577.724,E2 -1577.724} C_VEL
LIN {X 0,Y 739.284,Z 264.948,A -85,B 0,C 180,E1 -1580.126,E2 -1580.126} C_VEL
LIN {X 0,Y 739.253,Z 264.952,A -85,B 0,C 180,E1 -1581.984,E2 -1581.984} C_VEL
LIN {X 0,Y 739.297,Z 264.947,A -85,B 0,C 180,E1 -1584.026,E2 -1584.026} C_VEL
LIN {X 0,Y 739.324,Z 264.951,A -85,B 0,C 180,E1 -1586.484,E2 -1586.484} C_VEL
LIN {X 0,Y 739.319,Z 264.945,A -85,B 0,C 180,E1 -1589.229,E2 -1589.229} C_VEL
LIN {X 0,Y 739.313,Z 264.945,A -85,B 0,C 180,E1 -1591.724,E2 -1591.724} C_VEL
LIN {X 0,Y 739.349,Z 264.949,A -85,B 0,C 180,E1 -1594.164,E2 -1594.164} C_VEL
LIN {X 0,Y 739.319,Z 264.946,A -85,B 0,C 180,E1 -1596.781,E2 -1596.781} C_VEL
LIN {X 0,Y 739.343,Z 264.942,A -85,B 0,C 180,E1 -1598.899,E2 -1598.899} C_VEL
LIN {X 0,Y 739.346,Z 264.942,A -85,B 0,C 180,E1 -1601.332,E2 -1601.332} C_VEL
LIN {X 0,Y 739.34,Z 264.95,A -85,B 0,C 180,E1 -1604.053,E2 -1604.053} C_VEL
LIN {X 0,Y 739.315,Z 264.948,A -85,B 0,C 180,E1 -1606.299,E2 -1606.299} C_VEL
LIN {X 0,Y 739.334,Z 264.943,A -85,B 0,C 180,E1 -1608.524,E2 -1608.524} C_VEL
LIN {X 0,Y 739.375,Z 264.955,A -85,B 0,C 180,E1 -1610.576,E2 -1610.576} C_VEL
LIN {X 0,Y 739.764,Z 269.801,A -85,B 0,C 180,E1 -1611.149,E2 -1611.149} C_VEL
LIN {X 0,Y 739.628,Z 291.409,A -85,B 0,C 180,E1 -1613.625,E2 -1613.625} C_VEL
LIN {X 0,Y 739.49,Z 315.403,A -85,B 0,C 180,E1 -1616.334,E2 -1616.334} C_VEL
LIN {X 0,Y 739.428,Z 340.367,A -85,B 0,C 180,E1 -1619.118,E2 -1619.118} C_VEL
LIN {X 0,Y 739.853,Z 345.942,A -85,B 0,C 180,E1 -1619.186,E2 -1619.186} C_VEL
LIN {X 0,Y 739.67,Z 477.148,A -85,B 0,C 180,E1 -1620.475,E2 -1620.475} C_VEL
LIN {X 0,Y 739.647,Z 490.913,A -85,B 0,C 180,E1 -1620.712,E2 -1620.712} C_VEL
LIN {X 0,Y 739.601,Z 504.494,A -85,B 0,C 180,E1 -1621.051,E2 -1621.051} C_VEL
LIN {X 0,Y 739.497,Z 517.593,A -85,B 0,C 180,E1 -1621.493,E2 -1621.493} C_VEL
LIN {X 0,Y 739.454,Z 530.226,A -85,B 0,C 180,E1 -1622.036,E2 -1622.036} C_VEL
LIN {X 0,Y 739.41,Z 541.811,A -85,B 0,C 180,E1 -1622.647,E2 -1622.647} C_VEL
LIN {X 0,Y 739.322,Z 553.388,A -85,B 0,C 180,E1 -1623.395,E2 -1623.395} C_VEL
LIN {X 0,Y 739.292,Z 563.768,A -85,B 0,C 180,E1 -1624.211,E2 -1624.211} C_VEL
LIN {X 0,Y 739.262,Z 573.672,A -85,B 0,C 180,E1 -1625.164,E2 -1625.164} C_VEL
LIN {X 0,Y 739.214,Z 581.697,A -85,B 0,C 180,E1 -1626.119,E2 -1626.119} C_VEL
LIN {X 0,Y 739.183,Z 588.179,A -85,B 0,C 180,E1 -1627.076,E2 -1627.076} C_VEL
LIN {X 0,Y 739.147,Z 593.941,A -85,B 0,C 180,E1 -1628.172,E2 -1628.172} C_VEL
LIN {X 0,Y 739.175,Z 598.159,A -85,B 0,C 180,E1 -1629.27,E2 -1629.27} C_VEL
LIN {X 0,Y 739.145,Z 600.932,A -85,B 0,C 180,E1 -1630.373,E2 -1630.373} C_VEL
LIN {X 0,Y 739.138,Z 602.319,A -85,B 0,C 180,E1 -1631.479,E2 -1631.479} C_VEL
LIN {X 0,Y 739.155,Z 602.334,A -85,B 0,C 180,E1 -1632.589,E2 -1632.589} C_VEL
LIN {X 0,Y 739.13,Z 600.957,A -85,B 0,C 180,E1 -1633.705,E2 -1633.705} C_VEL
LIN {X 0,Y 739.187,Z 598.194,A -85,B 0,C 180,E1 -1634.806,E2 -1634.806} C_VEL
LIN {X 0,Y 738.561,Z 596.801,A -85,B 0,C 180,E1 -1635.248,E2 -1635.248} C_VEL
LIN {X 0,Y 735.696,Z 594.012,A -85,B 0,C 180,E1 -1635.954,E2 -1635.954} C_VEL
LIN {X 0,Y 733.249,Z 591.313,A -85,B 0,C 180,E1 -1636.508,E2 -1636.508} C_VEL
LIN {X 0,Y 732.194,Z 588.981,A -85,B 0,C 180,E1 -1636.927,E2 -1636.927} C_VEL
LIN {X 0,Y 732.108,Z 588.145,A -85,B 0,C 180,E1 -1637.068,E2 -1637.068} C_VEL
LIN {X 0,Y 732.153,Z 581.044,A -85,B 0,C 180,E1 -1638.115,E2 -1638.115} C_VEL
LIN {X 0,Y 732.171,Z 573.772,A -85,B 0,C 180,E1 -1638.982,E2 -1638.982} C_VEL
LIN {X 0,Y 732.224,Z 564.929,A -85,B 0,C 180,E1 -1639.852,E2 -1639.852} C_VEL
LIN {X 0,Y 732.302,Z 555.511,A -85,B 0,C 180,E1 -1640.623,E2 -1640.623} C_VEL
LIN {X 0,Y 732.369,Z 544.305,A -85,B 0,C 180,E1 -1641.385,E2 -1641.385} C_VEL
LIN {X 0,Y 732.427,Z 532.923,A -85,B 0,C 180,E1 -1642.019,E2 -1642.019} C_VEL
LIN {X 0,Y 732.471,Z 520.967,A -85,B 0,C 180,E1 -1642.563,E2 -1642.563} C_VEL
LIN {X 0,Y 732.61,Z 507.822,A -85,B 0,C 180,E1 -1643.042,E2 -1643.042} C_VEL
LIN {X 0,Y 732.674,Z 492.364,A -85,B 0,C 180,E1 -1643.456,E2 -1643.456} C_VEL
LIN {X 0,Y 732.719,Z 479.553,A -85,B 0,C 180,E1 -1643.691,E2 -1643.691} C_VEL
LIN {X 0,Y 732.73,Z 459.464,A -85,B 0,C 180,E1 -1643.915,E2 -1643.915} C_VEL
LIN {X 0,Y 732.732,Z 342.971,A -85,B 0,C 180,E1 -1645.06,E2 -1645.06} C_VEL
LIN {X 0,Y 732.352,Z 340.236,A -85,B 0,C 180,E1 -1645.114,E2 -1645.114} C_VEL
LIN {X 0,Y 732.462,Z 317.855,A -85,B 0,C 180,E1 -1647.633,E2 -1647.633} C_VEL
LIN {X 0,Y 732.599,Z 297.302,A -85,B 0,C 180,E1 -1649.971,E2 -1649.971} C_VEL
LIN {X 0,Y 732.778,Z 274.92,A -85,B 0,C 180,E1 -1652.552,E2 -1652.552} C_VEL
LIN {X 0,Y 732.669,Z 268.096,A -85,B 0,C 180,E1 -1653.347,E2 -1653.347} C_VEL
LIN {X 0,Y 732.274,Z 265.828,A -85,B 0,C 180,E1 -1653.628,E2 -1653.628} C_VEL
LIN {X 0,Y 732.254,Z 265.826,A -85,B 0,C 180,E1 -1655.697,E2 -1655.697} C_VEL
LIN {X 0,Y 732.286,Z 265.83,A -85,B 0,C 180,E1 -1658.339,E2 -1658.339} C_VEL
LIN {X 0,Y 732.278,Z 265.821,A -85,B 0,C 180,E1 -1660.916,E2 -1660.916} C_VEL
LIN {X 0,Y 732.253,Z 265.828,A -85,B 0,C 180,E1 -1663.529,E2 -1663.529} C_VEL
LIN {X 0,Y 732.251,Z 265.836,A -85,B 0,C 180,E1 -1665.842,E2 -1665.842} C_VEL
LIN {X 0,Y 732.27,Z 265.822,A -85,B 0,C 180,E1 -1668.698,E2 -1668.698} C_VEL
LIN {X 0,Y 732.272,Z 265.831,A -85,B 0,C 180,E1 -1671.662,E2 -1671.662} C_VEL
LIN {X 0,Y 732.242,Z 265.826,A -85,B 0,C 180,E1 -1674.399,E2 -1674.399} C_VEL
LIN {X 0,Y 732.264,Z 265.829,A -85,B 0,C 180,E1 -1676.959,E2 -1676.959} C_VEL
LIN {X 0,Y 732.263,Z 265.827,A -85,B 0,C 180,E1 -1679.537,E2 -1679.537} C_VEL
LIN {X 0,Y 732.252,Z 265.824,A -85,B 0,C 180,E1 -1682.048,E2 -1682.048} C_VEL
LIN {X 0,Y 732.267,Z 265.828,A -85,B 0,C 180,E1 -1684.503,E2 -1684.503} C_VEL
LIN {X 0,Y 732.271,Z 265.831,A -85,B 0,C 180,E1 -1686.909,E2 -1686.909} C_VEL
LIN {X 0,Y 732.289,Z 265.821,A -85,B 0,C 180,E1 -1689.272,E2 -1689.272} C_VEL
LIN {X 0,Y 732.297,Z 265.819,A -85,B 0,C 180,E1 -1691.599,E2 -1691.599} C_VEL
LIN {X 0,Y 732.306,Z 265.821,A -85,B 0,C 180,E1 -1693.895,E2 -1693.895} C_VEL
LIN {X 0,Y 732.277,Z 265.831,A -85,B 0,C 180,E1 -1696.164,E2 -1696.164} C_VEL
LIN {X 0,Y 732.284,Z 265.826,A -85,B 0,C 180,E1 -1698.411,E2 -1698.411} C_VEL
LIN {X 0,Y 732.323,Z 265.817,A -85,B 0,C 180,E1 -1700.641,E2 -1700.641} C_VEL
LIN {X 0,Y 732.303,Z 265.818,A -85,B 0,C 180,E1 -1702.856,E2 -1702.856} C_VEL
LIN {X 0,Y 732.336,Z 265.842,A -85,B 0,C 180,E1 -1705.129,E2 -1705.129} C_VEL
LIN {X 0,Y 732.261,Z 282.114,A -85,B 0,C 180,E1 -1707.532,E2 -1707.532} C_VEL
LIN {X 0,Y 732.273,Z 292.177,A -85,B 0,C 180,E1 -1709.005,E2 -1709.005} C_VEL
LIN {X 0,Y 732.885,Z 297.228,A -85,B 0,C 180,E1 -1709.075,E2 -1709.075} C_VEL
LIN {X 0,Y 732.71,Z 426.575,A -85,B 0,C 180,E1 -1710.358,E2 -1710.358} C_VEL
LIN {X 0,Y 732.689,Z 438.895,A -85,B 0,C 180,E1 -1710.564,E2 -1710.564} C_VEL
LIN {X 0,Y 732.618,Z 451.136,A -85,B 0,C 180,E1 -1710.855,E2 -1710.855} C_VEL
LIN {X 0,Y 732.512,Z 463.201,A -85,B 0,C 180,E1 -1711.231,E2 -1711.231} C_VEL
LIN {X 0,Y 732.507,Z 475.288,A -85,B 0,C 180,E1 -1711.711,E2 -1711.711} C_VEL
LIN {X 0,Y 732.41,Z 487.803,A -85,B 0,C 180,E1 -1712.328,E2 -1712.328} C_VEL
LIN {X 0,Y 732.313,Z 499.124,A -85,B 0,C 180,E1 -1713.014,E2 -1713.014} C_VEL
LIN {X 0,Y 732.29,Z 510.229,A -85,B 0,C 180,E1 -1713.838,E2 -1713.838} C_VEL
LIN {X 0,Y 732.172,Z 519.412,A -85,B 0,C 180,E1 -1714.663,E2 -1714.663} C_VEL
LIN {X 0,Y 732.125,Z 527.094,A -85,B 0,C 180,E1 -1715.489,E2 -1715.489} C_VEL
LIN {X 0,Y 732.14,Z 533.511,A -85,B 0,C 180,E1 -1716.315,E2 -1716.315} C_VEL
LIN {X 0,Y 732.101,Z 538.845,A -85,B 0,C 180,E1 -1717.143,E2 -1717.143} C_VEL
LIN {X 0,Y 732.075,Z 543.2,A -85,B 0,C 180,E1 -1717.973,E2 -1717.973} C_VEL
LIN {X 0,Y 732.093,Z 546.689,A -85,B 0,C 180,E1 -1718.804,E2 -1718.804} C_VEL
LIN {X 0,Y 732.062,Z 549.991,A -85,B 0,C 180,E1 -1719.916,E2 -1719.916} C_VEL
LIN {X 0,Y 732.036,Z 551.144,A -85,B 0,C 180,E1 -1720.473,E2 -1720.473} C_VEL
LIN {X 0,Y 732.062,Z 552.381,A -85,B 0,C 180,E1 -1721.59,E2 -1721.59} C_VEL
LIN {X 0,Y 732.078,Z 552.231,A -85,B 0,C 180,E1 -1722.711,E2 -1722.711} C_VEL
LIN {X 0,Y 732.029,Z 550.702,A -85,B 0,C 180,E1 -1723.838,E2 -1723.838} C_VEL
LIN {X 0,Y 732.085,Z 547.932,A -85,B 0,C 180,E1 -1724.906,E2 -1724.906} C_VEL
LIN {X 0,Y 732.088,Z 544.506,A -85,B 0,C 180,E1 -1725.822,E2 -1725.822} C_VEL
LIN {X 0,Y 732.112,Z 540.351,A -85,B 0,C 180,E1 -1726.678,E2 -1726.678} C_VEL
LIN {X 0,Y 732.111,Z 535.142,A -85,B 0,C 180,E1 -1727.539,E2 -1727.539} C_VEL
LIN {X 0,Y 732.136,Z 528.748,A -85,B 0,C 180,E1 -1728.402,E2 -1728.402} C_VEL
LIN {X 0,Y 732.185,Z 520.967,A -85,B 0,C 180,E1 -1729.27,E2 -1729.27} C_VEL
LIN {X 0,Y 732.231,Z 513.235,A -85,B 0,C 180,E1 -1729.996,E2 -1729.996} C_VEL
LIN {X 0,Y 732.315,Z 504.082,A -85,B 0,C 180,E1 -1730.724,E2 -1730.724} C_VEL
LIN {X 0,Y 732.368,Z 494.258,A -85,B 0,C 180,E1 -1731.383,E2 -1731.383} C_VEL
LIN {X 0,Y 732.42,Z 484.648,A -85,B 0,C 180,E1 -1731.928,E2 -1731.928} C_VEL
LIN {X 0,Y 732.47,Z 474.672,A -85,B 0,C 180,E1 -1732.406,E2 -1732.406} C_VEL
LIN {X 0,Y 732.535,Z 463.252,A -85,B 0,C 180,E1 -1732.856,E2 -1732.856} C_VEL
LIN {X 0,Y 732.629,Z 452.113,A -85,B 0,C 180,E1 -1733.209,E2 -1733.209} C_VEL
LIN {X 0,Y 732.664,Z 439.643,A -85,B 0,C 180,E1 -1733.512,E2 -1733.512} C_VEL
LIN {X 0,Y 732.703,Z 428.395,A -85,B 0,C 180,E1 -1733.708,E2 -1733.708} C_VEL
LIN {X 0,Y 732.759,Z 402.076,A -85,B 0,C 180,E1 -1733.987,E2 -1733.987} C_VEL
LIN {X 0,Y 732.808,Z 295.803,A -85,B 0,C 180,E1 -1735.031,E2 -1735.031} C_VEL
LIN {X 0,Y 732.264,Z 292.1,A -85,B 0,C 180,E1 -1735.096,E2 -1735.096} C_VEL
LIN {X 0,Y 732.306,Z 274.784,A -85,B 0,C 180,E1 -1737.637,E2 -1737.637} C_VEL
LIN {X 0,Y 732.284,Z 265.825,A -85,B 0,C 180,E1 -1738.98,E2 -1738.98} C_VEL
LIN {X 0,Y 732.234,Z 265.829,A -85,B 0,C 180,E1 -1741.64,E2 -1741.64} C_VEL
LIN {X 0,Y 732.251,Z 265.827,A -85,B 0,C 180,E1 -1743.695,E2 -1743.695} C_VEL
LIN {X 0,Y 732.232,Z 265.829,A -85,B 0,C 180,E1 -1745.696,E2 -1745.696} C_VEL
LIN {X 0,Y 732.272,Z 265.829,A -85,B 0,C 180,E1 -1748.339,E2 -1748.339} C_VEL
LIN {X 0,Y 732.264,Z 265.822,A -85,B 0,C 180,E1 -1750.916,E2 -1750.916} C_VEL
LIN {X 0,Y 732.237,Z 265.828,A -85,B 0,C 180,E1 -1753.528,E2 -1753.528} C_VEL
LIN {X 0,Y 732.277,Z 265.828,A -85,B 0,C 180,E1 -1755.837,E2 -1755.837} C_VEL
LIN {X 0,Y 732.279,Z 265.82,A -85,B 0,C 180,E1 -1758.7,E2 -1758.7} C_VEL
LIN {X 0,Y 732.278,Z 265.82,A -85,B 0,C 180,E1 -1760.853,E2 -1760.853} C_VEL
LIN {X 0,Y 732.236,Z 265.83,A -85,B 0,C 180,E1 -1763.465,E2 -1763.465} C_VEL
LIN {X 0,Y 732.266,Z 265.829,A -85,B 0,C 180,E1 -1765.642,E2 -1765.642} C_VEL
LIN {X 0,Y 732.262,Z 265.824,A -85,B 0,C 180,E1 -1768.258,E2 -1768.258} C_VEL
LIN {X 0,Y 732.254,Z 265.823,A -85,B 0,C 180,E1 -1770.801,E2 -1770.801} C_VEL
LIN {X 0,Y 732.238,Z 265.829,A -85,B 0,C 180,E1 -1773.282,E2 -1773.282} C_VEL
LIN {X 0,Y 732.254,Z 265.832,A -85,B 0,C 180,E1 -1775.712,E2 -1775.712} C_VEL
LIN {X 0,Y 732.265,Z 265.824,A -85,B 0,C 180,E1 -1778.096,E2 -1778.096} C_VEL
LIN {X 0,Y 732.26,Z 265.821,A -85,B 0,C 180,E1 -1780.44,E2 -1780.44} C_VEL
LIN {X 0,Y 732.268,Z 265.822,A -85,B 0,C 180,E1 -1782.751,E2 -1782.751} C_VEL
LIN {X 0,Y 732.301,Z 265.822,A -85,B 0,C 180,E1 -1785.034,E2 -1785.034} C_VEL
LIN {X 0,Y 732.284,Z 265.822,A -85,B 0,C 180,E1 -1787.852,E2 -1787.852} C_VEL
LIN {X 0,Y 732.295,Z 265.817,A -85,B 0,C 180,E1 -1790.117,E2 -1790.117} C_VEL
LIN {X 0,Y 732.306,Z 265.821,A -85,B 0,C 180,E1 -1792.857,E2 -1792.857} C_VEL
LIN {X 0,Y 732.339,Z 265.815,A -85,B 0,C 180,E1 -1795.612,E2 -1795.612} C_VEL
LIN {X 0,Y 732.298,Z 265.817,A -85,B 0,C 180,E1 -1798.356,E2 -1798.356} C_VEL
LIN {X 0,Y 732.241,Z 265.827,A -85,B 0,C 180,E1 -1800.548,E2 -1800.548} C_VEL
LIN {X 0,Y 732.288,Z 265.817,A -85,B 0,C 180,E1 -1802.193,E2 -1802.193} C_VEL
LIN {X 0,Y 732.334,Z 265.824,A -85,B 0,C 180,E1 -1804.938,E2 -1804.938} C_VEL
LIN {X 0,Y 732.31,Z 265.815,A -85,B 0,C 180,E1 -1807.696,E2 -1807.696} C_VEL
LIN {X 0,Y 732.291,Z 265.818,A -85,B 0,C 180,E1 -1809.914,E2 -1809.914} C_VEL
LIN {X 0,Y 732.299,Z 265.825,A -85,B 0,C 180,E1 -1812.685,E2 -1812.685} C_VEL
LIN {X 0,Y 732.306,Z 265.825,A -85,B 0,C 180,E1 -1814.98,E2 -1814.98} C_VEL
LIN {X 0,Y 732.285,Z 265.821,A -85,B 0,C 180,E1 -1817.249,E2 -1817.249} C_VEL
LIN {X 0,Y 732.264,Z 265.822,A -85,B 0,C 180,E1 -1819.56,E2 -1819.56} C_VEL
LIN {X 0,Y 732.265,Z 265.821,A -85,B 0,C 180,E1 -1821.904,E2 -1821.904} C_VEL
LIN {X 0,Y 732.269,Z 265.821,A -85,B 0,C 180,E1 -1823.687,E2 -1823.687} C_VEL
LIN {X 0,Y 732.259,Z 265.825,A -85,B 0,C 180,E1 -1826.105,E2 -1826.105} C_VEL
LIN {X 0,Y 732.284,Z 265.832,A -85,B 0,C 180,E1 -1828.572,E2 -1828.572} C_VEL
LIN {X 0,Y 732.274,Z 265.822,A -85,B 0,C 180,E1 -1831.1,E2 -1831.1} C_VEL
